LIN {X 0,Y 445.773,Z 444.898,A -85,B 0,C 180,E1 -8709.705,E2 -8709.705} C_VEL
LIN {X 0,Y 445.571,Z 450.254,A -85,B 0,C 180,E1 -8712.561,E2 -8712.561} C_VEL
LIN {X 0,Y 445.558,Z 452.75,A -85,B 0,C 180,E1 -8713.869,E2 -8713.869} C_VEL
LIN {X 0,Y 447.499,Z 463.216,A -85,B 0,C 180,E1 -8714.229,E2 -8714.229} C_VEL
LIN {X 0,Y 449.179,Z 473.492,A -85,B 0,C 180,E1 -8714.691,E2 -8714.691} C_VEL
LIN {X 0,Y 449.183,Z 481.574,A -85,B 0,C 180,E1 -8715.097,E2 -8715.097} C_VEL
LIN {X 0,Y 448.641,Z 491.717,A -85,B 0,C 180,E1 -8715.716,E2 -8715.716} C_VEL
LIN {X 0,Y 448.158,Z 500.718,A -85,B 0,C 180,E1 -8716.395,E2 -8716.395} C_VEL
LIN {X 0,Y 447.767,Z 508.998,A -85,B 0,C 180,E1 -8717.145,E2 -8717.145} C_VEL
LIN {X 0,Y 447.322,Z 516.853,A -85,B 0,C 180,E1 -8717.985,E2 -8717.985} C_VEL
LIN {X 0,Y 446.832,Z 524.074,A -85,B 0,C 180,E1 -8718.891,E2 -8718.891} C_VEL
LIN {X 0,Y 446.495,Z 530.28,A -85,B 0,C 180,E1 -8719.8,E2 -8719.8} C_VEL
LIN {X 0,Y 446.13,Z 536.82,A -85,B 0,C 180,E1 -8720.936,E2 -8720.936} C_VEL
LIN {X 0,Y 445.886,Z 541.323,A -85,B 0,C 180,E1 -8721.845,E2 -8721.845} C_VEL
LIN {X 0,Y 445.655,Z 546.972,A -85,B 0,C 180,E1 -8723.253,E2 -8723.253} C_VEL
LIN {X 0,Y 445.538,Z 551.142,A -85,B 0,C 180,E1 -8724.569,E2 -8724.569} C_VEL
LIN {X 0,Y 445.428,Z 553.506,A -85,B 0,C 180,E1 -8725.475,E2 -8725.475} C_VEL
LIN {X 0,Y 445.387,Z 555.304,A -85,B 0,C 180,E1 -8726.381,E2 -8726.381} C_VEL
LIN {X 0,Y 445.353,Z 557.747,A -85,B 0,C 180,E1 -8728.191,E2 -8728.191} C_VEL
LIN {X 0,Y 445.315,Z 558.334,A -85,B 0,C 180,E1 -8729.096,E2 -8729.096} C_VEL
LIN {X 0,Y 445.315,Z 558.334,A -85,B 0,C 180,E1 -8730.904,E2 -8730.904} C_VEL
LIN {X 0,Y 445.353,Z 557.747,A -85,B 0,C 180,E1 -8731.808,E2 -8731.808} C_VEL
LIN {X 0,Y 445.387,Z 555.305,A -85,B 0,C 180,E1 -8733.619,E2 -8733.619} C_VEL
LIN {X 0,Y 445.5,Z 552.359,A -85,B 0,C 180,E1 -8734.977,E2 -8734.977} C_VEL
LIN {X 0,Y 445.579,Z 548.371,A -85,B 0,C 180,E1 -8736.339,E2 -8736.339} C_VEL
LIN {X 0,Y 445.762,Z 543.24,A -85,B 0,C 180,E1 -8737.701,E2 -8737.701} C_VEL
LIN {X 0,Y 446.078,Z 537.978,A -85,B 0,C 180,E1 -8738.836,E2 -8738.836} C_VEL
LIN {X 0,Y 446.427,Z 531.659,A -85,B 0,C 180,E1 -8739.972,E2 -8739.972} C_VEL
LIN {X 0,Y 446.73,Z 525.704,A -85,B 0,C 180,E1 -8740.882,E2 -8740.882} C_VEL
LIN {X 0,Y 447.175,Z 518.775,A -85,B 0,C 180,E1 -8741.789,E2 -8741.789} C_VEL
LIN {X 0,Y 447.643,Z 510.591,A -85,B 0,C 180,E1 -8742.697,E2 -8742.697} C_VEL
LIN {X 0,Y 448.065,Z 502.329,A -85,B 0,C 180,E1 -8743.47,E2 -8743.47} C_VEL
LIN {X 0,Y 448.563,Z 493.356,A -85,B 0,C 180,E1 -8744.17,E2 -8744.17} C_VEL
LIN {X 0,Y 449.001,Z 484.602,A -85,B 0,C 180,E1 -8744.735,E2 -8744.735} C_VEL
LIN {X 0,Y 449.373,Z 474.797,A -85,B 0,C 180,E1 -8745.244,E2 -8745.244} C_VEL
LIN {X 0,Y 447.738,Z 464.356,A -85,B 0,C 180,E1 -8745.725,E2 -8745.725} C_VEL
LIN {X 0,Y 445.691,Z 453.752,A -85,B 0,C 180,E1 -8746.102,E2 -8746.102} C_VEL
LIN {X 0,Y 445.565,Z 452.689,A -85,B 0,C 180,E1 -8746.163,E2 -8746.163} C_VEL
LIN {X 0,Y 445.699,Z 446.656,A -85,B 0,C 180,E1 -8749.337,E2 -8749.337} C_VEL
LIN {X 0,Y 445.865,Z 441.314,A -85,B 0,C 180,E1 -8752.228,E2 -8752.228} C_VEL
LIN {X 0,Y 446.033,Z 436.032,A -85,B 0,C 180,E1 -8755.177,E2 -8755.177} C_VEL
LIN {X 0,Y 446.267,Z 430.816,A -85,B 0,C 180,E1 -8758.193,E2 -8758.193} C_VEL
LIN {X 0,Y 446.557,Z 424.849,A -85,B 0,C 180,E1 -8761.803,E2 -8761.803} C_VEL
LIN {X 0,Y 446.894,Z 419.658,A -85,B 0,C 180,E1 -8765.137,E2 -8765.137} C_VEL
LIN {X 0,Y 447.24,Z 415.135,A -85,B 0,C 180,E1 -8768.213,E2 -8768.213} C_VEL
LIN {X 0,Y 447.487,Z 410.971,A -85,B 0,C 180,E1 -8771.271,E2 -8771.271} C_VEL
LIN {X 0,Y 447.258,Z 407.884,A -85,B 0,C 180,E1 -8773.74,E2 -8773.74} C_VEL
LIN {X 0,Y 446.793,Z 404.867,A -85,B 0,C 180,E1 -8776.349,E2 -8776.349} C_VEL
LIN {X 0,Y 446.432,Z 402.428,A -85,B 0,C 180,E1 -8778.609,E2 -8778.609} C_VEL
LIN {X 0,Y 446.454,Z 402.376,A -85,B 0,C 180,E1 -8780.974,E2 -8780.974} C_VEL
LIN {X 0,Y 446.418,Z 402.379,A -85,B 0,C 180,E1 -8784.373,E2 -8784.373} C_VEL
LIN {X 0,Y 446.426,Z 402.372,A -85,B 0,C 180,E1 -8787.638,E2 -8787.638} C_VEL
LIN {X 0,Y 446.466,Z 402.374,A -85,B 0,C 180,E1 -8790.791,E2 -8790.791} C_VEL
LIN {X 0,Y 446.473,Z 402.366,A -85,B 0,C 180,E1 -8793.848,E2 -8793.848} C_VEL
LIN {X 0,Y 446.425,Z 402.379,A -85,B 0,C 180,E1 -8796.823,E2 -8796.823} C_VEL
LIN {X 0,Y 446.439,Z 402.37,A -85,B 0,C 180,E1 -8799.736,E2 -8799.736} C_VEL
LIN {X 0,Y 446.459,Z 402.375,A -85,B 0,C 180,E1 -8802.596,E2 -8802.596} C_VEL
LIN {X 0,Y 446.466,Z 402.367,A -85,B 0,C 180,E1 -8805.412,E2 -8805.412} C_VEL
LIN {X 0,Y 446.512,Z 402.364,A -85,B 0,C 180,E1 -8808.192,E2 -8808.192} C_VEL
LIN {X 0,Y 446.594,Z 402.352,A -85,B 0,C 180,E1 -8811.857,E2 -8811.857} C_VEL
LIN {X 0,Y 446.64,Z 402.352,A -85,B 0,C 180,E1 -8814.582,E2 -8814.582} C_VEL
LIN {X 0,Y 446.704,Z 402.337,A -85,B 0,C 180,E1 -8817.294,E2 -8817.294} C_VEL
LIN {X 0,Y 446.787,Z 402.33,A -85,B 0,C 180,E1 -8819.999,E2 -8819.999} C_VEL
LIN {X 0,Y 446.703,Z 402.341,A -85,B 0,C 180,E1 -8822.705,E2 -8822.705} C_VEL
LIN {X 0,Y 446.64,Z 402.353,A -85,B 0,C 180,E1 -8826.323,E2 -8826.323} C_VEL
LIN {X 0,Y 446.531,Z 402.359,A -85,B 0,C 180,E1 -8829.055,E2 -8829.055} C_VEL
LIN {X 0,Y 446.514,Z 402.363,A -85,B 0,C 180,E1 -8832.729,E2 -8832.729} C_VEL
LIN {X 0,Y 446.511,Z 402.368,A -85,B 0,C 180,E1 -8836.238,E2 -8836.238} C_VEL
LIN {X 0,Y 446.461,Z 402.368,A -85,B 0,C 180,E1 -8839.303,E2 -8839.303} C_VEL
LIN {X 0,Y 446.411,Z 402.379,A -85,B 0,C 180,E1 -8842.199,E2 -8842.199} C_VEL
LIN {X 0,Y 446.451,Z 402.369,A -85,B 0,C 180,E1 -8845.152,E2 -8845.152} C_VEL
LIN {X 0,Y 446.477,Z 402.37,A -85,B 0,C 180,E1 -8848.179,E2 -8848.179} C_VEL
LIN {X 0,Y 446.423,Z 402.373,A -85,B 0,C 180,E1 -8851.299,E2 -8851.299} C_VEL
LIN {X 0,Y 446.423,Z 402.373,A -85,B 0,C 180,E1 -8854.523,E2 -8854.523} C_VEL
LIN {X 0,Y 446.431,Z 402.375,A -85,B 0,C 180,E1 -8858.083,E2 -8858.083} C_VEL
LIN {X 0,Y 446.44,Z 402.37,A -85,B 0,C 180,E1 -8860.921,E2 -8860.921} C_VEL
LIN {X 0,Y 446.438,Z 402.376,A -85,B 0,C 180,E1 -8863.841,E2 -8863.841} C_VEL
LIN {X 0,Y 446.44,Z 402.371,A -85,B 0,C 180,E1 -8866.397,E2 -8866.397} C_VEL
LIN {X 0,Y 446.461,Z 402.373,A -85,B 0,C 180,E1 -8869.805,E2 -8869.805} C_VEL
LIN {X 0,Y 446.425,Z 402.374,A -85,B 0,C 180,E1 -8872.124,E2 -8872.124} C_VEL
LIN {X 0,Y 446.425,Z 402.379,A -85,B 0,C 180,E1 -8875.477,E2 -8875.477} C_VEL
LIN {X 0,Y 446.411,Z 402.374,A -85,B 0,C 180,E1 -8878.7,E2 -8878.7} C_VEL
LIN {X 0,Y 446.479,Z 402.368,A -85,B 0,C 180,E1 -8881.822,E2 -8881.822} C_VEL
LIN {X 0,Y 446.453,Z 402.37,A -85,B 0,C 180,E1 -8884.848,E2 -8884.848} C_VEL
LIN {X 0,Y 446.443,Z 402.37,A -85,B 0,C 180,E1 -8888.245,E2 -8888.245} C_VEL
LIN {X 0,Y 446.453,Z 402.374,A -85,B 0,C 180,E1 -8891.65,E2 -8891.65} C_VEL
LIN {X 0,Y 446.503,Z 402.366,A -85,B 0,C 180,E1 -8894.48,E2 -8894.48} C_VEL
LIN {X 0,Y 446.514,Z 402.363,A -85,B 0,C 180,E1 -8898.193,E2 -8898.193} C_VEL
LIN {X 0,Y 446.596,Z 402.355,A -85,B 0,C 180,E1 -8901.858,E2 -8901.858} C_VEL
LIN {X 0,Y 446.644,Z 402.349,A -85,B 0,C 180,E1 -8904.583,E2 -8904.583} C_VEL
LIN {X 0,Y 446.621,Z 402.353,A -85,B 0,C 180,E1 -8907.008,E2 -8907.008} C_VEL
LIN {X 0,Y 446.104,Z 402.421,A -85,B 0,C 180,E1 -8907.761,E2 -8907.761} C_VEL
LIN {X 0,Y 443.287,Z 402.776,A -85,B 0,C 180,E1 -8908.984,E2 -8908.984} C_VEL
LIN {X 0,Y 440.801,Z 403.085,A -85,B 0,C 180,E1 -8909.971,E2 -8909.971} C_VEL
LIN {X 0,Y 439.713,Z 403.216,A -85,B 0,C 180,E1 -8910.734,E2 -8910.734} C_VEL
LIN {X 0,Y 439.618,Z 403.225,A -85,B 0,C 180,E1 -8910.993,E2 -8910.993} C_VEL
LIN {X 0,Y 439.653,Z 403.222,A -85,B 0,C 180,E1 -8912.749,E2 -8912.749} C_VEL
LIN {X 0,Y 439.616,Z 403.227,A -85,B 0,C 180,E1 -8916.425,E2 -8916.425} C_VEL
LIN {X 0,Y 439.497,Z 403.241,A -85,B 0,C 180,E1 -8919.202,E2 -8919.202} C_VEL
LIN {X 0,Y 439.462,Z 403.247,A -85,B 0,C 180,E1 -8922.938,E2 -8922.938} C_VEL
LIN {X 0,Y 439.444,Z 403.247,A -85,B 0,C 180,E1 -8926.349,E2 -8926.349} C_VEL
LIN {X 0,Y 439.399,Z 403.248,A -85,B 0,C 180,E1 -8929.626,E2 -8929.626} C_VEL
LIN {X 0,Y 439.361,Z 403.259,A -85,B 0,C 180,E1 -8932.575,E2 -8932.575} C_VEL
LIN {X 0,Y 439.401,Z 403.247,A -85,B 0,C 180,E1 -8935.585,E2 -8935.585} C_VEL
LIN {X 0,Y 439.413,Z 403.252,A -85,B 0,C 180,E1 -8938.674,E2 -8938.674} C_VEL
LIN {X 0,Y 439.366,Z 403.253,A -85,B 0,C 180,E1 -8942.031,E2 -8942.031} C_VEL
LIN {X 0,Y 439.392,Z 403.248,A -85,B 0,C 180,E1 -8945.341,E2 -8945.341} C_VEL
LIN {X 0,Y 439.391,Z 403.253,A -85,B 0,C 180,E1 -8948.594,E2 -8948.594} C_VEL
LIN {X 0,Y 439.4,Z 403.247,A -85,B 0,C 180,E1 -8951.259,E2 -8951.259} C_VEL
LIN {X 0,Y 439.404,Z 403.249,A -85,B 0,C 180,E1 -8954.728,E2 -8954.728} C_VEL
LIN {X 0,Y 439.391,Z 403.25,A -85,B 0,C 180,E1 -8957.796,E2 -8957.796} C_VEL
LIN {X 0,Y 439.431,Z 403.251,A -85,B 0,C 180,E1 -8960.229,E2 -8960.229} C_VEL
LIN {X 0,Y 439.372,Z 403.253,A -85,B 0,C 180,E1 -8963.713,E2 -8963.713} C_VEL
LIN {X 0,Y 439.37,Z 403.251,A -85,B 0,C 180,E1 -8967.055,E2 -8967.055} C_VEL
LIN {X 0,Y 439.392,Z 403.253,A -85,B 0,C 180,E1 -8970.276,E2 -8970.276} C_VEL
LIN {X 0,Y 439.428,Z 403.246,A -85,B 0,C 180,E1 -8973.589,E2 -8973.589} C_VEL
LIN {X 0,Y 439.382,Z 403.252,A -85,B 0,C 180,E1 -8976.43,E2 -8976.43} C_VEL
LIN {X 0,Y 439.383,Z 403.251,A -85,B 0,C 180,E1 -8979.397,E2 -8979.397} C_VEL
LIN {X 0,Y 439.428,Z 403.246,A -85,B 0,C 180,E1 -8982.31,E2 -8982.31} C_VEL
LIN {X 0,Y 439.447,Z 403.242,A -85,B 0,C 180,E1 -8985.175,E2 -8985.175} C_VEL
LIN {X 0,Y 439.479,Z 403.242,A -85,B 0,C 180,E1 -8988.002,E2 -8988.002} C_VEL
LIN {X 0,Y 439.544,Z 403.237,A -85,B 0,C 180,E1 -8991.727,E2 -8991.727} C_VEL
LIN {X 0,Y 439.617,Z 403.22,A -85,B 0,C 180,E1 -8994.496,E2 -8994.496} C_VEL
LIN {X 0,Y 439.632,Z 403.22,A -85,B 0,C 180,E1 -8998.168,E2 -8998.168} C_VEL
LIN {X 0,Y 439.76,Z 403.205,A -85,B 0,C 180,E1 -9000.001,E2 -9000.001} C_VEL
LIN {X 0,Y 439.653,Z 403.216,A -85,B 0,C 180,E1 -9002.749,E2 -9002.749} C_VEL
LIN {X 0,Y 439.615,Z 403.22,A -85,B 0,C 180,E1 -9006.426,E2 -9006.426} C_VEL
LIN {X 0,Y 439.497,Z 403.239,A -85,B 0,C 180,E1 -9009.202,E2 -9009.202} C_VEL
LIN {X 0,Y 439.463,Z 403.241,A -85,B 0,C 180,E1 -9012.938,E2 -9012.938} C_VEL
LIN {X 0,Y 439.445,Z 403.241,A -85,B 0,C 180,E1 -9016.349,E2 -9016.349} C_VEL
LIN {X 0,Y 439.4,Z 403.251,A -85,B 0,C 180,E1 -9019.627,E2 -9019.627} C_VEL
LIN {X 0,Y 439.363,Z 403.252,A -85,B 0,C 180,E1 -9022.576,E2 -9022.576} C_VEL
LIN {X 0,Y 439.404,Z 403.25,A -85,B 0,C 180,E1 -9025.585,E2 -9025.585} C_VEL
LIN {X 0,Y 439.416,Z 403.247,A -85,B 0,C 180,E1 -9028.674,E2 -9028.674} C_VEL
LIN {X 0,Y 439.369,Z 403.251,A -85,B 0,C 180,E1 -9032.031,E2 -9032.031} C_VEL
LIN {X 0,Y 439.396,Z 403.255,A -85,B 0,C 180,E1 -9035.341,E2 -9035.341} C_VEL
LIN {X 0,Y 439.388,Z 403.256,A -85,B 0,C 180,E1 -9038.595,E2 -9038.595} C_VEL
LIN {X 0,Y 439.381,Z 403.257,A -85,B 0,C 180,E1 -9040.981,E2 -9040.981} C_VEL
LIN {X 0,Y 439.869,Z 406.467,A -85,B 0,C 180,E1 -9044.03,E2 -9044.03} C_VEL
LIN {X 0,Y 440.286,Z 409.495,A -85,B 0,C 180,E1 -9046.656,E2 -9046.656} C_VEL
LIN {X 0,Y 440.456,Z 412.609,A -85,B 0,C 180,E1 -9049.141,E2 -9049.141} C_VEL
LIN {X 0,Y 440.258,Z 415.779,A -85,B 0,C 180,E1 -9051.496,E2 -9051.496} C_VEL
LIN {X 0,Y 439.849,Z 420.662,A -85,B 0,C 180,E1 -9054.886,E2 -9054.886} C_VEL
LIN {X 0,Y 439.508,Z 425.659,A -85,B 0,C 180,E1 -9058.151,E2 -9058.151} C_VEL
LIN {X 0,Y 439.238,Z 430.761,A -85,B 0,C 180,E1 -9061.314,E2 -9061.314} C_VEL
LIN {X 0,Y 438.999,Z 435.948,A -85,B 0,C 180,E1 -9064.39,E2 -9064.39} C_VEL
LIN {X 0,Y 438.794,Z 441.194,A -85,B 0,C 180,E1 -9067.394,E2 -9067.394} C_VEL
LIN {X 0,Y 438.627,Z 446.502,A -85,B 0,C 180,E1 -9070.338,E2 -9070.338} C_VEL
LIN {X 0,Y 438.486,Z 452.562,A -85,B 0,C 180,E1 -9073.599,E2 -9073.599} C_VEL
LIN {X 0,Y 440.489,Z 462.989,A -85,B 0,C 180,E1 -9073.971,E2 -9073.971} C_VEL
LIN {X 0,Y 442.142,Z 473.275,A -85,B 0,C 180,E1 -9074.441,E2 -9074.441} C_VEL
LIN {X 0,Y 442.414,Z 478.317,A -85,B 0,C 180,E1 -9074.687,E2 -9074.687} C_VEL
LIN {X 0,Y 441.855,Z 489.873,A -85,B 0,C 180,E1 -9075.374,E2 -9075.374} C_VEL
LIN {X 0,Y 441.347,Z 499.155,A -85,B 0,C 180,E1 -9076.063,E2 -9076.063} C_VEL
LIN {X 0,Y 440.915,Z 507.557,A -85,B 0,C 180,E1 -9076.815,E2 -9076.815} C_VEL
LIN {X 0,Y 440.353,Z 516.641,A -85,B 0,C 180,E1 -9077.792,E2 -9077.792} C_VEL
LIN {X 0,Y 439.828,Z 523.862,A -85,B 0,C 180,E1 -9078.712,E2 -9078.712} C_VEL
LIN {X 0,Y 439.478,Z 530.068,A -85,B 0,C 180,E1 -9079.636,E2 -9079.636} C_VEL
LIN {X 0,Y 439.085,Z 536.608,A -85,B 0,C 180,E1 -9080.79,E2 -9080.79} C_VEL
LIN {X 0,Y 438.832,Z 541.111,A -85,B 0,C 180,E1 -9081.713,E2 -9081.713} C_VEL
LIN {X 0,Y 438.591,Z 546.604,A -85,B 0,C 180,E1 -9083.097,E2 -9083.097} C_VEL
LIN {X 0,Y 438.439,Z 550.929,A -85,B 0,C 180,E1 -9084.481,E2 -9084.481} C_VEL
LIN {X 0,Y 438.357,Z 553.295,A -85,B 0,C 180,E1 -9085.402,E2 -9085.402} C_VEL
LIN {X 0,Y 438.332,Z 556.48,A -85,B 0,C 180,E1 -9087.243,E2 -9087.243} C_VEL
LIN {X 0,Y 438.275,Z 557.536,A -85,B 0,C 180,E1 -9088.162,E2 -9088.162} C_VEL
LIN {X 0,Y 438.231,Z 558.123,A -85,B 0,C 180,E1 -9089.081,E2 -9089.081} C_VEL
LIN {X 0,Y 438.23,Z 558.123,A -85,B 0,C 180,E1 -9090.919,E2 -9090.919} C_VEL
LIN {X 0,Y 438.275,Z 557.537,A -85,B 0,C 180,E1 -9091.838,E2 -9091.838} C_VEL
LIN {X 0,Y 438.289,Z 555.093,A -85,B 0,C 180,E1 -9093.677,E2 -9093.677} C_VEL
LIN {X 0,Y 438.414,Z 552.147,A -85,B 0,C 180,E1 -9095.058,E2 -9095.058} C_VEL
LIN {X 0,Y 438.507,Z 548.159,A -85,B 0,C 180,E1 -9096.441,E2 -9096.441} C_VEL
LIN {X 0,Y 438.717,Z 543.029,A -85,B 0,C 180,E1 -9097.826,E2 -9097.826} C_VEL
LIN {X 0,Y 439.038,Z 537.766,A -85,B 0,C 180,E1 -9098.979,E2 -9098.979} C_VEL
LIN {X 0,Y 439.4,Z 531.447,A -85,B 0,C 180,E1 -9100.133,E2 -9100.133} C_VEL
LIN {X 0,Y 439.717,Z 525.492,A -85,B 0,C 180,E1 -9101.057,E2 -9101.057} C_VEL
LIN {X 0,Y 440.212,Z 518.563,A -85,B 0,C 180,E1 -9101.978,E2 -9101.978} C_VEL
LIN {X 0,Y 440.697,Z 510.379,A -85,B 0,C 180,E1 -9102.9,E2 -9102.9} C_VEL
LIN {X 0,Y 441.159,Z 501.795,A -85,B 0,C 180,E1 -9103.713,E2 -9103.713} C_VEL
LIN {X 0,Y 441.655,Z 493.144,A -85,B 0,C 180,E1 -9104.397,E2 -9104.397} C_VEL
LIN {X 0,Y 442.161,Z 483.382,A -85,B 0,C 180,E1 -9105.027,E2 -9105.027} C_VEL
LIN {X 0,Y 442.497,Z 475.874,A -85,B 0,C 180,E1 -9105.428,E2 -9105.428} C_VEL
LIN {X 0,Y 440.758,Z 464.605,A -85,B 0,C 180,E1 -9105.964,E2 -9105.964} C_VEL
LIN {X 0,Y 438.726,Z 454.283,A -85,B 0,C 180,E1 -9106.348,E2 -9106.348} C_VEL
LIN {X 0,Y 438.49,Z 452.559,A -85,B 0,C 180,E1 -9106.402,E2 -9106.402} C_VEL
LIN {X 0,Y 438.625,Z 446.5,A -85,B 0,C 180,E1 -9109.662,E2 -9109.662} C_VEL
LIN {X 0,Y 438.793,Z 441.188,A -85,B 0,C 180,E1 -9112.606,E2 -9112.606} C_VEL
LIN {X 0,Y 438.998,Z 435.939,A -85,B 0,C 180,E1 -9115.61,E2 -9115.61} C_VEL
LIN {X 0,Y 439.236,Z 430.751,A -85,B 0,C 180,E1 -9118.686,E2 -9118.686} C_VEL
LIN {X 0,Y 439.527,Z 425.322,A -85,B 0,C 180,E1 -9122.062,E2 -9122.062} C_VEL
LIN {X 0,Y 439.849,Z 420.656,A -85,B 0,C 180,E1 -9125.114,E2 -9125.114} C_VEL
LIN {X 0,Y 440.244,Z 415.74,A -85,B 0,C 180,E1 -9128.534,E2 -9128.534} C_VEL
LIN {X 0,Y 440.459,Z 411.885,A -85,B 0,C 180,E1 -9131.415,E2 -9131.415} C_VEL
LIN {X 0,Y 440.2,Z 408.622,A -85,B 0,C 180,E1 -9134.073,E2 -9134.073} C_VEL
LIN {X 0,Y 439.669,Z 405.005,A -85,B 0,C 180,E1 -9137.331,E2 -9137.331} C_VEL
LIN {X 0,Y 439.379,Z 403.257,A -85,B 0,C 180,E1 -9139.019,E2 -9139.019} C_VEL
LIN {X 0,Y 439.382,Z 403.256,A -85,B 0,C 180,E1 -9141.605,E2 -9141.605} C_VEL
LIN {X 0,Y 439.398,Z 403.255,A -85,B 0,C 180,E1 -9144.843,E2 -9144.843} C_VEL
LIN {X 0,Y 439.386,Z 403.249,A -85,B 0,C 180,E1 -9148.14,E2 -9148.14} C_VEL
LIN {X 0,Y 439.421,Z 403.246,A -85,B 0,C 180,E1 -9151.326,E2 -9151.326} C_VEL
LIN {X 0,Y 439.401,Z 403.25,A -85,B 0,C 180,E1 -9154.414,E2 -9154.414} C_VEL
LIN {X 0,Y 439.36,Z 403.253,A -85,B 0,C 180,E1 -9157.424,E2 -9157.424} C_VEL
LIN {X 0,Y 439.436,Z 403.25,A -85,B 0,C 180,E1 -9160.662,E2 -9160.662} C_VEL
LIN {X 0,Y 439.457,Z 403.243,A -85,B 0,C 180,E1 -9164.224,E2 -9164.224} C_VEL
LIN {X 0,Y 439.478,Z 403.239,A -85,B 0,C 180,E1 -9168.001,E2 -9168.001} C_VEL
LIN {X 0,Y 439.542,Z 403.23,A -85,B 0,C 180,E1 -9171.726,E2 -9171.726} C_VEL
LIN {X 0,Y 439.615,Z 403.228,A -85,B 0,C 180,E1 -9174.495,E2 -9174.495} C_VEL
LIN {X 0,Y 439.63,Z 403.223,A -85,B 0,C 180,E1 -9178.167,E2 -9178.167} C_VEL
LIN {X 0,Y 439.757,Z 403.206,A -85,B 0,C 180,E1 -9179.999,E2 -9179.999} C_VEL
LIN {X 0,Y 439.65,Z 403.219,A -85,B 0,C 180,E1 -9182.748,E2 -9182.748} C_VEL
LIN {X 0,Y 439.611,Z 403.227,A -85,B 0,C 180,E1 -9186.425,E2 -9186.425} C_VEL
LIN {X 0,Y 439.493,Z 403.235,A -85,B 0,C 180,E1 -9189.201,E2 -9189.201} C_VEL
LIN {X 0,Y 439.458,Z 403.24,A -85,B 0,C 180,E1 -9192.937,E2 -9192.937} C_VEL
LIN {X 0,Y 439.453,Z 403.245,A -85,B 0,C 180,E1 -9196.354,E2 -9196.354} C_VEL
LIN {X 0,Y 439.395,Z 403.25,A -85,B 0,C 180,E1 -9199.626,E2 -9199.626} C_VEL
LIN {X 0,Y 439.358,Z 403.254,A -85,B 0,C 180,E1 -9202.575,E2 -9202.575} C_VEL
LIN {X 0,Y 439.398,Z 403.25,A -85,B 0,C 180,E1 -9205.585,E2 -9205.585} C_VEL
LIN {X 0,Y 439.418,Z 403.245,A -85,B 0,C 180,E1 -9208.673,E2 -9208.673} C_VEL
LIN {X 0,Y 439.376,Z 403.256,A -85,B 0,C 180,E1 -9212.033,E2 -9212.033} C_VEL
LIN {X 0,Y 439.389,Z 403.25,A -85,B 0,C 180,E1 -9215.341,E2 -9215.341} C_VEL
LIN {X 0,Y 439.392,Z 403.248,A -85,B 0,C 180,E1 -9218.593,E2 -9218.593} C_VEL
LIN {X 0,Y 439.398,Z 403.249,A -85,B 0,C 180,E1 -9221.259,E2 -9221.259} C_VEL
LIN {X 0,Y 439.403,Z 403.247,A -85,B 0,C 180,E1 -9224.728,E2 -9224.728} C_VEL
LIN {X 0,Y 439.406,Z 403.252,A -85,B 0,C 180,E1 -9227.798,E2 -9227.798} C_VEL
LIN {X 0,Y 439.443,Z 403.243,A -85,B 0,C 180,E1 -9230.23,E2 -9230.23} C_VEL
LIN {X 0,Y 439.371,Z 403.256,A -85,B 0,C 180,E1 -9233.713,E2 -9233.713} C_VEL
LIN {X 0,Y 439.366,Z 403.254,A -85,B 0,C 180,E1 -9237.054,E2 -9237.054} C_VEL
LIN {X 0,Y 439.377,Z 403.25,A -85,B 0,C 180,E1 -9240.274,E2 -9240.274} C_VEL
LIN {X 0,Y 439.425,Z 403.252,A -85,B 0,C 180,E1 -9243.397,E2 -9243.397} C_VEL
LIN {X 0,Y 439.381,Z 403.249,A -85,B 0,C 180,E1 -9246.43,E2 -9246.43} C_VEL
LIN {X 0,Y 439.385,Z 403.256,A -85,B 0,C 180,E1 -9249.397,E2 -9249.397} C_VEL
LIN {X 0,Y 439.427,Z 403.247,A -85,B 0,C 180,E1 -9252.31,E2 -9252.31} C_VEL
LIN {X 0,Y 439.443,Z 403.249,A -85,B 0,C 180,E1 -9255.174,E2 -9255.174} C_VEL
LIN {X 0,Y 439.48,Z 403.239,A -85,B 0,C 180,E1 -9258.002,E2 -9258.002} C_VEL
LIN {X 0,Y 439.544,Z 403.234,A -85,B 0,C 180,E1 -9261.727,E2 -9261.727} C_VEL
LIN {X 0,Y 439.619,Z 403.224,A -85,B 0,C 180,E1 -9264.496,E2 -9264.496} C_VEL
LIN {X 0,Y 439.633,Z 403.222,A -85,B 0,C 180,E1 -9268.168,E2 -9268.168} C_VEL
LIN {X 0,Y 439.761,Z 403.207,A -85,B 0,C 180,E1 -9270,E2 -9270} C_VEL
LIN {X 0,Y 439.618,Z 403.225,A -85,B 0,C 180,E1 -9270.993,E2 -9270.993} C_VEL
LIN {X 0,Y 438.903,Z 403.313,A -85,B 0,C 180,E1 -9271.758,E2 -9271.758} C_VEL
LIN {X 0,Y 435.924,Z 403.686,A -85,B 0,C 180,E1 -9272.997,E2 -9272.997} C_VEL
LIN {X 0,Y 433.473,Z 403.991,A -85,B 0,C 180,E1 -9273.997,E2 -9273.997} C_VEL
LIN {X 0,Y 432.5,Z 404.113,A -85,B 0,C 180,E1 -9274.771,E2 -9274.771} C_VEL
LIN {X 0,Y 432.463,Z 404.114,A -85,B 0,C 180,E1 -9275.033,E2 -9275.033} C_VEL
LIN {X 0,Y 432.582,Z 404.101,A -85,B 0,C 180,E1 -9277.679,E2 -9277.679} C_VEL
LIN {X 0,Y 432.39,Z 404.125,A -85,B 0,C 180,E1 -9281.247,E2 -9281.247} C_VEL
LIN {X 0,Y 432.37,Z 404.127,A -85,B 0,C 180,E1 -9284.112,E2 -9284.112} C_VEL
LIN {X 0,Y 432.394,Z 404.127,A -85,B 0,C 180,E1 -9287.012,E2 -9287.012} C_VEL
LIN {X 0,Y 432.335,Z 404.128,A -85,B 0,C 180,E1 -9289.961,E2 -9289.961} C_VEL
LIN {X 0,Y 432.315,Z 404.133,A -85,B 0,C 180,E1 -9292.964,E2 -9292.964} C_VEL
LIN {X 0,Y 432.36,Z 404.125,A -85,B 0,C 180,E1 -9296.032,E2 -9296.032} C_VEL
LIN {X 0,Y 432.339,Z 404.128,A -85,B 0,C 180,E1 -9299.187,E2 -9299.187} C_VEL
LIN {X 0,Y 432.319,Z 404.136,A -85,B 0,C 180,E1 -9302.443,E2 -9302.443} C_VEL
LIN {X 0,Y 432.341,Z 404.127,A -85,B 0,C 180,E1 -9305.632,E2 -9305.632} C_VEL
LIN {X 0,Y 432.353,Z 404.129,A -85,B 0,C 180,E1 -9308.717,E2 -9308.717} C_VEL
LIN {X 0,Y 432.369,Z 404.124,A -85,B 0,C 180,E1 -9311.792,E2 -9311.792} C_VEL
LIN {X 0,Y 432.374,Z 404.13,A -85,B 0,C 180,E1 -9314.342,E2 -9314.342} C_VEL
LIN {X 0,Y 432.329,Z 404.135,A -85,B 0,C 180,E1 -9318.203,E2 -9318.203} C_VEL
LIN {X 0,Y 432.348,Z 404.126,A -85,B 0,C 180,E1 -9321.284,E2 -9321.284} C_VEL
LIN {X 0,Y 432.34,Z 404.131,A -85,B 0,C 180,E1 -9324.368,E2 -9324.368} C_VEL
LIN {X 0,Y 432.323,Z 404.13,A -85,B 0,C 180,E1 -9327.558,E2 -9327.558} C_VEL
LIN {X 0,Y 432.39,Z 404.124,A -85,B 0,C 180,E1 -9329.744,E2 -9329.744} C_VEL
LIN {X 0,Y 432.395,Z 404.121,A -85,B 0,C 180,E1 -9333.373,E2 -9333.373} C_VEL
LIN {X 0,Y 432.367,Z 404.13,A -85,B 0,C 180,E1 -9336.024,E2 -9336.024} C_VEL
LIN {X 0,Y 432.345,Z 404.126,A -85,B 0,C 180,E1 -9339.046,E2 -9339.046} C_VEL
LIN {X 0,Y 432.374,Z 404.128,A -85,B 0,C 180,E1 -9342.012,E2 -9342.012} C_VEL
LIN {X 0,Y 432.397,Z 404.119,A -85,B 0,C 180,E1 -9344.927,E2 -9344.927} C_VEL
LIN {X 0,Y 432.455,Z 404.12,A -85,B 0,C 180,E1 -9347.804,E2 -9347.804} C_VEL
LIN {X 0,Y 432.488,Z 404.114,A -85,B 0,C 180,E1 -9351.591,E2 -9351.591} C_VEL
LIN {X 0,Y 432.594,Z 404.096,A -85,B 0,C 180,E1 -9354.407,E2 -9354.407} C_VEL
LIN {X 0,Y 432.602,Z 404.096,A -85,B 0,C 180,E1 -9358.139,E2 -9358.139} C_VEL
LIN {X 0,Y 432.73,Z 404.081,A -85,B 0,C 180,E1 -9360.001,E2 -9360.001} C_VEL
LIN {X 0,Y 432.602,Z 404.094,A -85,B 0,C 180,E1 -9362.794,E2 -9362.794} C_VEL
LIN {X 0,Y 432.569,Z 404.098,A -85,B 0,C 180,E1 -9366.531,E2 -9366.531} C_VEL
LIN {X 0,Y 432.44,Z 404.12,A -85,B 0,C 180,E1 -9369.354,E2 -9369.354} C_VEL
LIN {X 0,Y 432.428,Z 404.117,A -85,B 0,C 180,E1 -9372.804,E2 -9372.804} C_VEL
LIN {X 0,Y 432.41,Z 404.118,A -85,B 0,C 180,E1 -9376.48,E2 -9376.48} C_VEL
LIN {X 0,Y 432.336,Z 404.128,A -85,B 0,C 180,E1 -9379.961,E2 -9379.961} C_VEL
LIN {X 0,Y 432.317,Z 404.133,A -85,B 0,C 180,E1 -9382.965,E2 -9382.965} C_VEL
LIN {X 0,Y 432.363,Z 404.124,A -85,B 0,C 180,E1 -9386.033,E2 -9386.033} C_VEL
LIN {X 0,Y 432.341,Z 404.134,A -85,B 0,C 180,E1 -9389.188,E2 -9389.188} C_VEL
LIN {X 0,Y 432.322,Z 404.13,A -85,B 0,C 180,E1 -9392.444,E2 -9392.444} C_VEL
LIN {X 0,Y 432.345,Z 404.131,A -85,B 0,C 180,E1 -9395.633,E2 -9395.633} C_VEL
LIN {X 0,Y 432.351,Z 404.132,A -85,B 0,C 180,E1 -9398.717,E2 -9398.717} C_VEL
LIN {X 0,Y 432.326,Z 404.135,A -85,B 0,C 180,E1 -9400.561,E2 -9400.561} C_VEL
LIN {X 0,Y 432.728,Z 406.574,A -85,B 0,C 180,E1 -9403.043,E2 -9403.043} C_VEL
LIN {X 0,Y 433.178,Z 409.587,A -85,B 0,C 180,E1 -9405.762,E2 -9405.762} C_VEL
LIN {X 0,Y 433.43,Z 412.673,A -85,B 0,C 180,E1 -9408.333,E2 -9408.333} C_VEL
LIN {X 0,Y 433.279,Z 415.81,A -85,B 0,C 180,E1 -9410.758,E2 -9410.758} C_VEL
LIN {X 0,Y 432.873,Z 420.713,A -85,B 0,C 180,E1 -9414.271,E2 -9414.271} C_VEL
LIN {X 0,Y 432.504,Z 425.776,A -85,B 0,C 180,E1 -9417.67,E2 -9417.67} C_VEL
LIN {X 0,Y 432.213,Z 430.694,A -85,B 0,C 180,E1 -9420.803,E2 -9420.803} C_VEL
LIN {X 0,Y 431.979,Z 435.85,A -85,B 0,C 180,E1 -9423.943,E2 -9423.943} C_VEL
LIN {X 0,Y 431.741,Z 441.072,A -85,B 0,C 180,E1 -9427.003,E2 -9427.003} C_VEL
LIN {X 0,Y 431.554,Z 446.345,A -85,B 0,C 180,E1 -9430.002,E2 -9430.002} C_VEL
LIN {X 0,Y 431.399,Z 452.353,A -85,B 0,C 180,E1 -9433.309,E2 -9433.309} C_VEL
LIN {X 0,Y 434.13,Z 467.212,A -85,B 0,C 180,E1 -9433.883,E2 -9433.883} C_VEL
LIN {X 0,Y 435.564,Z 478.106,A -85,B 0,C 180,E1 -9434.44,E2 -9434.44} C_VEL
LIN {X 0,Y 434.956,Z 489.661,A -85,B 0,C 180,E1 -9435.137,E2 -9435.137} C_VEL
LIN {X 0,Y 434.434,Z 498.943,A -85,B 0,C 180,E1 -9435.837,E2 -9435.837} C_VEL
LIN {X 0,Y 433.916,Z 508.134,A -85,B 0,C 180,E1 -9436.681,E2 -9436.681} C_VEL
LIN {X 0,Y 433.398,Z 516.429,A -85,B 0,C 180,E1 -9437.593,E2 -9437.593} C_VEL
LIN {X 0,Y 432.844,Z 523.65,A -85,B 0,C 180,E1 -9438.527,E2 -9438.527} C_VEL
LIN {X 0,Y 432.468,Z 529.855,A -85,B 0,C 180,E1 -9439.466,E2 -9439.466} C_VEL
LIN {X 0,Y 432.059,Z 536.396,A -85,B 0,C 180,E1 -9440.638,E2 -9440.638} C_VEL
LIN {X 0,Y 431.791,Z 540.899,A -85,B 0,C 180,E1 -9441.576,E2 -9441.576} C_VEL
LIN {X 0,Y 431.522,Z 546.393,A -85,B 0,C 180,E1 -9442.984,E2 -9442.984} C_VEL
LIN {X 0,Y 431.343,Z 550.717,A -85,B 0,C 180,E1 -9444.39,E2 -9444.39} C_VEL
LIN {X 0,Y 431.288,Z 553.084,A -85,B 0,C 180,E1 -9445.326,E2 -9445.326} C_VEL
LIN {X 0,Y 431.229,Z 556.269,A -85,B 0,C 180,E1 -9447.197,E2 -9447.197} C_VEL
LIN {X 0,Y 431.2,Z 557.326,A -85,B 0,C 180,E1 -9448.132,E2 -9448.132} C_VEL
LIN {X 0,Y 431.149,Z 557.912,A -85,B 0,C 180,E1 -9449.066,E2 -9449.066} C_VEL
LIN {X 0,Y 431.149,Z 557.913,A -85,B 0,C 180,E1 -9450.934,E2 -9450.934} C_VEL
LIN {X 0,Y 431.2,Z 557.326,A -85,B 0,C 180,E1 -9451.868,E2 -9451.868} C_VEL
LIN {X 0,Y 431.196,Z 554.881,A -85,B 0,C 180,E1 -9453.738,E2 -9453.738} C_VEL
LIN {X 0,Y 431.329,Z 551.936,A -85,B 0,C 180,E1 -9455.141,E2 -9455.141} C_VEL
LIN {X 0,Y 431.442,Z 547.948,A -85,B 0,C 180,E1 -9456.547,E2 -9456.547} C_VEL
LIN {X 0,Y 431.646,Z 542.816,A -85,B 0,C 180,E1 -9457.955,E2 -9457.955} C_VEL
LIN {X 0,Y 431.973,Z 537.553,A -85,B 0,C 180,E1 -9459.127,E2 -9459.127} C_VEL
LIN {X 0,Y 432.362,Z 531.234,A -85,B 0,C 180,E1 -9460.3,E2 -9460.3} C_VEL
LIN {X 0,Y 432.717,Z 525.279,A -85,B 0,C 180,E1 -9461.238,E2 -9461.238} C_VEL
LIN {X 0,Y 433.251,Z 518.352,A -85,B 0,C 180,E1 -9462.174,E2 -9462.174} C_VEL
LIN {X 0,Y 433.76,Z 510.168,A -85,B 0,C 180,E1 -9463.11,E2 -9463.11} C_VEL
LIN {X 0,Y 434.222,Z 501.992,A -85,B 0,C 180,E1 -9463.901,E2 -9463.901} C_VEL
LIN {X 0,Y 434.742,Z 492.931,A -85,B 0,C 180,E1 -9464.631,E2 -9464.631} C_VEL
LIN {X 0,Y 435.284,Z 483.17,A -85,B 0,C 180,E1 -9465.27,E2 -9465.27} C_VEL
LIN {X 0,Y 435.602,Z 476.949,A -85,B 0,C 180,E1 -9465.618,E2 -9465.618} C_VEL
LIN {X 0,Y 433.76,Z 464.865,A -85,B 0,C 180,E1 -9466.213,E2 -9466.213} C_VEL
LIN {X 0,Y 431.558,Z 453.706,A -85,B 0,C 180,E1 -9466.636,E2 -9466.636} C_VEL
LIN {X 0,Y 431.4,Z 452.356,A -85,B 0,C 180,E1 -9466.689,E2 -9466.689} C_VEL
LIN {X 0,Y 431.552,Z 446.344,A -85,B 0,C 180,E1 -9469.998,E2 -9469.998} C_VEL
LIN {X 0,Y 431.74,Z 441.067,A -85,B 0,C 180,E1 -9472.996,E2 -9472.996} C_VEL
LIN {X 0,Y 431.976,Z 435.842,A -85,B 0,C 180,E1 -9476.057,E2 -9476.057} C_VEL
LIN {X 0,Y 432.201,Z 430.687,A -85,B 0,C 180,E1 -9479.197,E2 -9479.197} C_VEL
LIN {X 0,Y 432.511,Z 425.624,A -85,B 0,C 180,E1 -9482.426,E2 -9482.426} C_VEL
LIN {X 0,Y 432.874,Z 420.656,A -85,B 0,C 180,E1 -9485.766,E2 -9485.766} C_VEL
LIN {X 0,Y 433.241,Z 416.325,A -85,B 0,C 180,E1 -9488.862,E2 -9488.862} C_VEL
LIN {X 0,Y 433.421,Z 412.553,A -85,B 0,C 180,E1 -9491.763,E2 -9491.763} C_VEL
LIN {X 0,Y 433.15,Z 409.35,A -85,B 0,C 180,E1 -9494.445,E2 -9494.445} C_VEL
LIN {X 0,Y 432.703,Z 406.549,A -85,B 0,C 180,E1 -9496.986,E2 -9496.986} C_VEL
LIN {X 0,Y 432.324,Z 404.134,A -85,B 0,C 180,E1 -9499.439,E2 -9499.439} C_VEL
LIN {X 0,Y 432.344,Z 404.131,A -85,B 0,C 180,E1 -9501.85,E2 -9501.85} C_VEL
LIN {X 0,Y 432.338,Z 404.134,A -85,B 0,C 180,E1 -9505.322,E2 -9505.322} C_VEL
LIN {X 0,Y 432.331,Z 404.132,A -85,B 0,C 180,E1 -9508.654,E2 -9508.654} C_VEL
LIN {X 0,Y 432.38,Z 404.122,A -85,B 0,C 180,E1 -9511.876,E2 -9511.876} C_VEL
LIN {X 0,Y 432.347,Z 404.13,A -85,B 0,C 180,E1 -9514.998,E2 -9514.998} C_VEL
LIN {X 0,Y 432.352,Z 404.126,A -85,B 0,C 180,E1 -9518.045,E2 -9518.045} C_VEL
LIN {X 0,Y 432.381,Z 404.125,A -85,B 0,C 180,E1 -9521.029,E2 -9521.029} C_VEL
LIN {X 0,Y 432.425,Z 404.117,A -85,B 0,C 180,E1 -9523.96,E2 -9523.96} C_VEL
LIN {X 0,Y 432.453,Z 404.113,A -85,B 0,C 180,E1 -9527.803,E2 -9527.803} C_VEL
LIN {X 0,Y 432.486,Z 404.108,A -85,B 0,C 180,E1 -9531.59,E2 -9531.59} C_VEL
LIN {X 0,Y 432.592,Z 404.102,A -85,B 0,C 180,E1 -9534.406,E2 -9534.406} C_VEL
LIN {X 0,Y 432.6,Z 404.098,A -85,B 0,C 180,E1 -9538.138,E2 -9538.138} C_VEL
LIN {X 0,Y 432.727,Z 404.081,A -85,B 0,C 180,E1 -9539.999,E2 -9539.999} C_VEL
LIN {X 0,Y 432.599,Z 404.097,A -85,B 0,C 180,E1 -9542.793,E2 -9542.793} C_VEL
LIN {X 0,Y 432.566,Z 404.103,A -85,B 0,C 180,E1 -9546.53,E2 -9546.53} C_VEL
LIN {X 0,Y 432.436,Z 404.115,A -85,B 0,C 180,E1 -9549.353,E2 -9549.353} C_VEL
LIN {X 0,Y 432.423,Z 404.117,A -85,B 0,C 180,E1 -9552.803,E2 -9552.803} C_VEL
LIN {X 0,Y 432.415,Z 404.12,A -85,B 0,C 180,E1 -9556.483,E2 -9556.483} C_VEL
LIN {X 0,Y 432.331,Z 404.134,A -85,B 0,C 180,E1 -9559.96,E2 -9559.96} C_VEL
LIN {X 0,Y 432.312,Z 404.13,A -85,B 0,C 180,E1 -9562.964,E2 -9562.964} C_VEL
LIN {X 0,Y 432.358,Z 404.132,A -85,B 0,C 180,E1 -9566.032,E2 -9566.032} C_VEL
LIN {X 0,Y 432.345,Z 404.126,A -85,B 0,C 180,E1 -9569.187,E2 -9569.187} C_VEL
LIN {X 0,Y 432.324,Z 404.131,A -85,B 0,C 180,E1 -9572.295,E2 -9572.295} C_VEL
LIN {X 0,Y 432.333,Z 404.128,A -85,B 0,C 180,E1 -9574.677,E2 -9574.677} C_VEL
LIN {X 0,Y 432.346,Z 404.129,A -85,B 0,C 180,E1 -9578.148,E2 -9578.148} C_VEL
LIN {X 0,Y 432.366,Z 404.129,A -85,B 0,C 180,E1 -9581.608,E2 -9581.608} C_VEL
LIN {X 0,Y 432.371,Z 404.124,A -85,B 0,C 180,E1 -9584.342,E2 -9584.342} C_VEL
LIN {X 0,Y 432.359,Z 404.125,A -85,B 0,C 180,E1 -9587.009,E2 -9587.009} C_VEL
LIN {X 0,Y 432.35,Z 404.13,A -85,B 0,C 180,E1 -9589.817,E2 -9589.817} C_VEL
LIN {X 0,Y 432.31,Z 404.132,A -85,B 0,C 180,E1 -9593.023,E2 -9593.023} C_VEL
LIN {X 0,Y 432.354,Z 404.127,A -85,B 0,C 180,E1 -9595.997,E2 -9595.997} C_VEL
LIN {X 0,Y 432.342,Z 404.134,A -85,B 0,C 180,E1 -9599.49,E2 -9599.49} C_VEL
LIN {X 0,Y 432.388,Z 404.123,A -85,B 0,C 180,E1 -9602.929,E2 -9602.929} C_VEL
LIN {X 0,Y 432.366,Z 404.124,A -85,B 0,C 180,E1 -9606.024,E2 -9606.024} C_VEL
LIN {X 0,Y 432.346,Z 404.13,A -85,B 0,C 180,E1 -9609.046,E2 -9609.046} C_VEL
LIN {X 0,Y 432.374,Z 404.126,A -85,B 0,C 180,E1 -9612.011,E2 -9612.011} C_VEL
LIN {X 0,Y 432.391,Z 404.127,A -85,B 0,C 180,E1 -9614.927,E2 -9614.927} C_VEL
LIN {X 0,Y 432.455,Z 404.115,A -85,B 0,C 180,E1 -9617.804,E2 -9617.804} C_VEL
LIN {X 0,Y 432.488,Z 404.113,A -85,B 0,C 180,E1 -9621.591,E2 -9621.591} C_VEL
LIN {X 0,Y 432.595,Z 404.099,A -85,B 0,C 180,E1 -9624.406,E2 -9624.406} C_VEL
LIN {X 0,Y 432.603,Z 404.097,A -85,B 0,C 180,E1 -9628.138,E2 -9628.138} C_VEL
LIN {X 0,Y 432.73,Z 404.083,A -85,B 0,C 180,E1 -9630,E2 -9630} C_VEL
LIN {X 0,Y 432.602,Z 404.1,A -85,B 0,C 180,E1 -9632.794,E2 -9632.794} C_VEL
LIN {X 0,Y 432.463,Z 404.114,A -85,B 0,C 180,E1 -9635.033,E2 -9635.033} C_VEL
LIN {X 0,Y 431.904,Z 404.185,A -85,B 0,C 180,E1 -9635.812,E2 -9635.812} C_VEL
LIN {X 0,Y 429.057,Z 404.542,A -85,B 0,C 180,E1 -9637.077,E2 -9637.077} C_VEL
LIN {X 0,Y 426.572,Z 404.85,A -85,B 0,C 180,E1 -9638.098,E2 -9638.098} C_VEL
LIN {X 0,Y 425.49,Z 404.987,A -85,B 0,C 180,E1 -9638.888,E2 -9638.888} C_VEL
LIN {X 0,Y 425.399,Z 404.995,A -85,B 0,C 180,E1 -9639.156,E2 -9639.156} C_VEL
LIN {X 0,Y 425.39,Z 405,A -85,B 0,C 180,E1 -9642.904,E2 -9642.904} C_VEL
LIN {X 0,Y 425.358,Z 405.003,A -85,B 0,C 180,E1 -9646.605,E2 -9646.605} C_VEL
LIN {X 0,Y 425.325,Z 405.002,A -85,B 0,C 180,E1 -9649.636,E2 -9649.636} C_VEL
LIN {X 0,Y 425.303,Z 405.004,A -85,B 0,C 180,E1 -9653.365,E2 -9653.365} C_VEL
LIN {X 0,Y 425.345,Z 405.002,A -85,B 0,C 180,E1 -9656.845,E2 -9656.845} C_VEL
LIN {X 0,Y 425.287,Z 405.005,A -85,B 0,C 180,E1 -9659.72,E2 -9659.72} C_VEL
LIN {X 0,Y 425.278,Z 405.008,A -85,B 0,C 180,E1 -9663.048,E2 -9663.048} C_VEL
LIN {X 0,Y 425.281,Z 405.008,A -85,B 0,C 180,E1 -9665.929,E2 -9665.929} C_VEL
LIN {X 0,Y 425.306,Z 405.004,A -85,B 0,C 180,E1 -9669.046,E2 -9669.046} C_VEL
LIN {X 0,Y 425.327,Z 405.004,A -85,B 0,C 180,E1 -9672.646,E2 -9672.646} C_VEL
LIN {X 0,Y 425.29,Z 405.005,A -85,B 0,C 180,E1 -9675.282,E2 -9675.282} C_VEL
LIN {X 0,Y 425.27,Z 405.01,A -85,B 0,C 180,E1 -9678.622,E2 -9678.622} C_VEL
LIN {X 0,Y 425.31,Z 405.002,A -85,B 0,C 180,E1 -9681.103,E2 -9681.103} C_VEL
LIN {X 0,Y 425.295,Z 405.006,A -85,B 0,C 180,E1 -9684.664,E2 -9684.664} C_VEL
LIN {X 0,Y 425.269,Z 405.015,A -85,B 0,C 180,E1 -9688.074,E2 -9688.074} C_VEL
LIN {X 0,Y 425.333,Z 405,A -85,B 0,C 180,E1 -9691.369,E2 -9691.369} C_VEL
LIN {X 0,Y 425.291,Z 405.006,A -85,B 0,C 180,E1 -9694.555,E2 -9694.555} C_VEL
LIN {X 0,Y 425.283,Z 405.009,A -85,B 0,C 180,E1 -9697.662,E2 -9697.662} C_VEL
LIN {X 0,Y 425.357,Z 404.997,A -85,B 0,C 180,E1 -9700.704,E2 -9700.704} C_VEL
LIN {X 0,Y 425.394,Z 404.997,A -85,B 0,C 180,E1 -9703.689,E2 -9703.689} C_VEL
LIN {X 0,Y 425.407,Z 404.995,A -85,B 0,C 180,E1 -9707.599,E2 -9707.599} C_VEL
LIN {X 0,Y 425.438,Z 404.99,A -85,B 0,C 180,E1 -9711.45,E2 -9711.45} C_VEL
LIN {X 0,Y 425.55,Z 404.974,A -85,B 0,C 180,E1 -9714.314,E2 -9714.314} C_VEL
LIN {X 0,Y 425.572,Z 404.972,A -85,B 0,C 180,E1 -9718.108,E2 -9718.108} C_VEL
LIN {X 0,Y 425.699,Z 404.957,A -85,B 0,C 180,E1 -9720.001,E2 -9720.001} C_VEL
LIN {X 0,Y 425.554,Z 404.972,A -85,B 0,C 180,E1 -9722.84,E2 -9722.84} C_VEL
LIN {X 0,Y 425.528,Z 404.975,A -85,B 0,C 180,E1 -9726.639,E2 -9726.639} C_VEL
LIN {X 0,Y 425.398,Z 404.998,A -85,B 0,C 180,E1 -9729.51,E2 -9729.51} C_VEL
LIN {X 0,Y 425.391,Z 404.994,A -85,B 0,C 180,E1 -9732.904,E2 -9732.904} C_VEL
LIN {X 0,Y 425.359,Z 404.997,A -85,B 0,C 180,E1 -9736.606,E2 -9736.606} C_VEL
LIN {X 0,Y 425.326,Z 405.004,A -85,B 0,C 180,E1 -9739.636,E2 -9739.636} C_VEL
LIN {X 0,Y 425.305,Z 405.009,A -85,B 0,C 180,E1 -9743.366,E2 -9743.366} C_VEL
LIN {X 0,Y 425.346,Z 405.001,A -85,B 0,C 180,E1 -9746.845,E2 -9746.845} C_VEL
LIN {X 0,Y 425.29,Z 405.006,A -85,B 0,C 180,E1 -9749.72,E2 -9749.72} C_VEL
LIN {X 0,Y 425.281,Z 405.013,A -85,B 0,C 180,E1 -9753.049,E2 -9753.049} C_VEL
LIN {X 0,Y 425.284,Z 405.009,A -85,B 0,C 180,E1 -9755.93,E2 -9755.93} C_VEL
LIN {X 0,Y 425.3,Z 405.011,A -85,B 0,C 180,E1 -9759.044,E2 -9759.044} C_VEL
LIN {X 0,Y 425.33,Z 405.23,A -85,B 0,C 180,E1 -9760.529,E2 -9760.529} C_VEL
LIN {X 0,Y 425.83,Z 408.662,A -85,B 0,C 180,E1 -9763.883,E2 -9763.883} C_VEL
LIN {X 0,Y 426.258,Z 411.566,A -85,B 0,C 180,E1 -9766.507,E2 -9766.507} C_VEL
LIN {X 0,Y 426.383,Z 414.966,A -85,B 0,C 180,E1 -9769.307,E2 -9769.307} C_VEL
LIN {X 0,Y 426.075,Z 419.058,A -85,B 0,C 180,E1 -9772.389,E2 -9772.389} C_VEL
LIN {X 0,Y 425.681,Z 423.945,A -85,B 0,C 180,E1 -9775.852,E2 -9775.852} C_VEL
LIN {X 0,Y 425.297,Z 429.024,A -85,B 0,C 180,E1 -9779.238,E2 -9779.238} C_VEL
LIN {X 0,Y 425.025,Z 434.039,A -85,B 0,C 180,E1 -9782.42,E2 -9782.42} C_VEL
LIN {X 0,Y 424.778,Z 439.212,A -85,B 0,C 180,E1 -9785.567,E2 -9785.567} C_VEL
LIN {X 0,Y 424.592,Z 444.453,A -85,B 0,C 180,E1 -9788.645,E2 -9788.645} C_VEL
LIN {X 0,Y 424.367,Z 449.712,A -85,B 0,C 180,E1 -9791.66,E2 -9791.66} C_VEL
LIN {X 0,Y 424.329,Z 452.422,A -85,B 0,C 180,E1 -9793.048,E2 -9793.048} C_VEL
LIN {X 0,Y 426.272,Z 462.585,A -85,B 0,C 180,E1 -9793.423,E2 -9793.423} C_VEL
LIN {X 0,Y 428.062,Z 472.839,A -85,B 0,C 180,E1 -9793.915,E2 -9793.915} C_VEL
LIN {X 0,Y 428.657,Z 478.922,A -85,B 0,C 180,E1 -9794.244,E2 -9794.244} C_VEL
LIN {X 0,Y 428.082,Z 489.449,A -85,B 0,C 180,E1 -9794.893,E2 -9794.893} C_VEL
LIN {X 0,Y 427.54,Z 498.731,A -85,B 0,C 180,E1 -9795.604,E2 -9795.604} C_VEL
LIN {X 0,Y 427.059,Z 506.726,A -85,B 0,C 180,E1 -9796.335,E2 -9796.335} C_VEL
LIN {X 0,Y 426.591,Z 514.297,A -85,B 0,C 180,E1 -9797.149,E2 -9797.149} C_VEL
LIN {X 0,Y 425.872,Z 523.438,A -85,B 0,C 180,E1 -9798.337,E2 -9798.337} C_VEL
LIN {X 0,Y 425.454,Z 529.643,A -85,B 0,C 180,E1 -9799.29,E2 -9799.29} C_VEL
LIN {X 0,Y 425.025,Z 536.184,A -85,B 0,C 180,E1 -9800.482,E2 -9800.482} C_VEL
LIN {X 0,Y 424.737,Z 540.687,A -85,B 0,C 180,E1 -9801.436,E2 -9801.436} C_VEL
LIN {X 0,Y 424.44,Z 546.18,A -85,B 0,C 180,E1 -9802.866,E2 -9802.866} C_VEL
LIN {X 0,Y 424.252,Z 550.505,A -85,B 0,C 180,E1 -9804.296,E2 -9804.296} C_VEL
LIN {X 0,Y 424.219,Z 552.873,A -85,B 0,C 180,E1 -9805.248,E2 -9805.248} C_VEL
LIN {X 0,Y 424.126,Z 556.057,A -85,B 0,C 180,E1 -9807.15,E2 -9807.15} C_VEL
LIN {X 0,Y 424.126,Z 557.115,A -85,B 0,C 180,E1 -9808.101,E2 -9808.101} C_VEL
LIN {X 0,Y 424.07,Z 557.702,A -85,B 0,C 180,E1 -9809.05,E2 -9809.05} C_VEL
LIN {X 0,Y 424.07,Z 557.702,A -85,B 0,C 180,E1 -9810.949,E2 -9810.949} C_VEL
LIN {X 0,Y 424.126,Z 557.115,A -85,B 0,C 180,E1 -9811.899,E2 -9811.899} C_VEL
LIN {X 0,Y 424.108,Z 554.67,A -85,B 0,C 180,E1 -9813.8,E2 -9813.8} C_VEL
LIN {X 0,Y 424.246,Z 551.724,A -85,B 0,C 180,E1 -9815.227,E2 -9815.227} C_VEL
LIN {X 0,Y 424.361,Z 547.735,A -85,B 0,C 180,E1 -9816.657,E2 -9816.657} C_VEL
LIN {X 0,Y 424.59,Z 542.604,A -85,B 0,C 180,E1 -9818.088,E2 -9818.088} C_VEL
LIN {X 0,Y 424.925,Z 537.341,A -85,B 0,C 180,E1 -9819.28,E2 -9819.28} C_VEL
LIN {X 0,Y 425.336,Z 531.021,A -85,B 0,C 180,E1 -9820.472,E2 -9820.472} C_VEL
LIN {X 0,Y 425.732,Z 525.067,A -85,B 0,C 180,E1 -9821.425,E2 -9821.425} C_VEL
LIN {X 0,Y 426.3,Z 518.14,A -85,B 0,C 180,E1 -9822.375,E2 -9822.375} C_VEL
LIN {X 0,Y 426.822,Z 509.955,A -85,B 0,C 180,E1 -9823.327,E2 -9823.327} C_VEL
LIN {X 0,Y 427.339,Z 501.171,A -85,B 0,C 180,E1 -9824.184,E2 -9824.184} C_VEL
LIN {X 0,Y 427.871,Z 492.72,A -85,B 0,C 180,E1 -9824.871,E2 -9824.871} C_VEL
LIN {X 0,Y 428.441,Z 482.959,A -85,B 0,C 180,E1 -9825.52,E2 -9825.52} C_VEL
LIN {X 0,Y 428.572,Z 476.731,A -85,B 0,C 180,E1 -9825.881,E2 -9825.881} C_VEL
LIN {X 0,Y 426.631,Z 464.259,A -85,B 0,C 180,E1 -9826.505,E2 -9826.505} C_VEL
LIN {X 0,Y 424.479,Z 453.446,A -85,B 0,C 180,E1 -9826.922,E2 -9826.922} C_VEL
LIN {X 0,Y 424.317,Z 452.163,A -85,B 0,C 180,E1 -9826.981,E2 -9826.981} C_VEL
LIN {X 0,Y 424.505,Z 446.189,A -85,B 0,C 180,E1 -9830.344,E2 -9830.344} C_VEL
LIN {X 0,Y 424.679,Z 440.94,A -85,B 0,C 180,E1 -9833.401,E2 -9833.401} C_VEL
LIN {X 0,Y 424.968,Z 435.38,A -85,B 0,C 180,E1 -9836.742,E2 -9836.742} C_VEL
LIN {X 0,Y 425.188,Z 430.627,A -85,B 0,C 180,E1 -9839.727,E2 -9839.727} C_VEL
LIN {X 0,Y 425.509,Z 425.589,A -85,B 0,C 180,E1 -9843.027,E2 -9843.027} C_VEL
LIN {X 0,Y 425.851,Z 421.235,A -85,B 0,C 180,E1 -9846.033,E2 -9846.033} C_VEL
LIN {X 0,Y 426.254,Z 416.913,A -85,B 0,C 180,E1 -9849.201,E2 -9849.201} C_VEL
LIN {X 0,Y 426.375,Z 413.193,A -85,B 0,C 180,E1 -9852.119,E2 -9852.119} C_VEL
LIN {X 0,Y 426.06,Z 410.07,A -85,B 0,C 180,E1 -9854.821,E2 -9854.821} C_VEL
LIN {X 0,Y 425.523,Z 406.683,A -85,B 0,C 180,E1 -9858.006,E2 -9858.006} C_VEL
LIN {X 0,Y 425.288,Z 405.012,A -85,B 0,C 180,E1 -9859.872,E2 -9859.872} C_VEL
LIN {X 0,Y 425.282,Z 405.012,A -85,B 0,C 180,E1 -9862.486,E2 -9862.486} C_VEL
LIN {X 0,Y 425.305,Z 405.005,A -85,B 0,C 180,E1 -9865.817,E2 -9865.817} C_VEL
LIN {X 0,Y 425.302,Z 405.006,A -85,B 0,C 180,E1 -9869.235,E2 -9869.235} C_VEL
LIN {X 0,Y 425.346,Z 405.001,A -85,B 0,C 180,E1 -9872.442,E2 -9872.442} C_VEL
LIN {X 0,Y 425.347,Z 404.998,A -85,B 0,C 180,E1 -9875.601,E2 -9875.601} C_VEL
LIN {X 0,Y 425.288,Z 405.012,A -85,B 0,C 180,E1 -9878.681,E2 -9878.681} C_VEL
LIN {X 0,Y 425.328,Z 405,A -85,B 0,C 180,E1 -9881.702,E2 -9881.702} C_VEL
LIN {X 0,Y 425.344,Z 405.005,A -85,B 0,C 180,E1 -9884.67,E2 -9884.67} C_VEL
LIN {X 0,Y 425.406,Z 404.99,A -85,B 0,C 180,E1 -9887.598,E2 -9887.598} C_VEL
LIN {X 0,Y 425.436,Z 404.987,A -85,B 0,C 180,E1 -9891.449,E2 -9891.449} C_VEL
LIN {X 0,Y 425.548,Z 404.978,A -85,B 0,C 180,E1 -9894.313,E2 -9894.313} C_VEL
LIN {X 0,Y 425.569,Z 404.974,A -85,B 0,C 180,E1 -9898.107,E2 -9898.107} C_VEL
LIN {X 0,Y 425.696,Z 404.957,A -85,B 0,C 180,E1 -9899.999,E2 -9899.999} C_VEL
LIN {X 0,Y 425.551,Z 404.974,A -85,B 0,C 180,E1 -9902.839,E2 -9902.839} C_VEL
LIN {X 0,Y 425.524,Z 404.979,A -85,B 0,C 180,E1 -9906.638,E2 -9906.638} C_VEL
LIN {X 0,Y 425.394,Z 404.992,A -85,B 0,C 180,E1 -9909.509,E2 -9909.509} C_VEL
LIN {X 0,Y 425.386,Z 404.993,A -85,B 0,C 180,E1 -9912.903,E2 -9912.903} C_VEL
LIN {X 0,Y 425.363,Z 404.998,A -85,B 0,C 180,E1 -9916.609,E2 -9916.609} C_VEL
LIN {X 0,Y 425.321,Z 405.003,A -85,B 0,C 180,E1 -9919.635,E2 -9919.635} C_VEL
LIN {X 0,Y 425.3,Z 405.004,A -85,B 0,C 180,E1 -9923.365,E2 -9923.365} C_VEL
LIN {X 0,Y 425.341,Z 404.999,A -85,B 0,C 180,E1 -9926.844,E2 -9926.844} C_VEL
LIN {X 0,Y 425.311,Z 405.007,A -85,B 0,C 180,E1 -9929.717,E2 -9929.717} C_VEL
LIN {X 0,Y 425.277,Z 405.007,A -85,B 0,C 180,E1 -9933.048,E2 -9933.048} C_VEL
LIN {X 0,Y 425.277,Z 405.013,A -85,B 0,C 180,E1 -9935.929,E2 -9935.929} C_VEL
LIN {X 0,Y 425.306,Z 405.003,A -85,B 0,C 180,E1 -9939.046,E2 -9939.046} C_VEL
LIN {X 0,Y 425.325,Z 405.001,A -85,B 0,C 180,E1 -9942.646,E2 -9942.646} C_VEL
LIN {X 0,Y 425.312,Z 405.005,A -85,B 0,C 180,E1 -9946.052,E2 -9946.052} C_VEL
LIN {X 0,Y 425.303,Z 405.003,A -85,B 0,C 180,E1 -9948.626,E2 -9948.626} C_VEL
LIN {X 0,Y 425.315,Z 405.004,A -85,B 0,C 180,E1 -9951.104,E2 -9951.104} C_VEL
LIN {X 0,Y 425.294,Z 405.004,A -85,B 0,C 180,E1 -9954.664,E2 -9954.664} C_VEL
LIN {X 0,Y 425.259,Z 405.01,A -85,B 0,C 180,E1 -9958.073,E2 -9958.073} C_VEL
LIN {X 0,Y 425.326,Z 405.007,A -85,B 0,C 180,E1 -9961.368,E2 -9961.368} C_VEL
LIN {X 0,Y 425.29,Z 405.005,A -85,B 0,C 180,E1 -9964.555,E2 -9964.555} C_VEL
LIN {X 0,Y 425.283,Z 405.009,A -85,B 0,C 180,E1 -9967.662,E2 -9967.662} C_VEL
LIN {X 0,Y 425.357,Z 404.998,A -85,B 0,C 180,E1 -9970.704,E2 -9970.704} C_VEL
LIN {X 0,Y 425.384,Z 404.998,A -85,B 0,C 180,E1 -9973.689,E2 -9973.689} C_VEL
LIN {X 0,Y 425.408,Z 404.994,A -85,B 0,C 180,E1 -9977.598,E2 -9977.598} C_VEL
LIN {X 0,Y 425.439,Z 404.992,A -85,B 0,C 180,E1 -9981.45,E2 -9981.45} C_VEL
LIN {X 0,Y 425.552,Z 404.976,A -85,B 0,C 180,E1 -9984.314,E2 -9984.314} C_VEL
LIN {X 0,Y 425.572,Z 404.973,A -85,B 0,C 180,E1 -9988.107,E2 -9988.107} C_VEL
LIN {X 0,Y 425.7,Z 404.959,A -85,B 0,C 180,E1 -9990,E2 -9990} C_VEL
LIN {X 0,Y 425.554,Z 404.978,A -85,B 0,C 180,E1 -9992.84,E2 -9992.84} C_VEL
LIN {X 0,Y 425.529,Z 404.981,A -85,B 0,C 180,E1 -9996.639,E2 -9996.639} C_VEL
LIN {X 0,Y 425.399,Z 404.995,A -85,B 0,C 180,E1 -9999.156,E2 -9999.156} C_VEL
LIN {X 0,Y 424.728,Z 405.081,A -85,B 0,C 180,E1 -9999.946,E2 -9999.946} C_VEL
LIN {X 0,Y 421.879,Z 405.438,A -85,B 0,C 180,E1 -10001.229,E2 -10001.229} C_VEL
LIN {X 0,Y 419.463,Z 405.739,A -85,B 0,C 180,E1 -10002.265,E2 -10002.265} C_VEL
LIN {X 0,Y 418.412,Z 405.869,A -85,B 0,C 180,E1 -10003.066,E2 -10003.066} C_VEL
LIN {X 0,Y 418.318,Z 405.878,A -85,B 0,C 180,E1 -10003.337,E2 -10003.337} C_VEL
LIN {X 0,Y 418.309,Z 405.882,A -85,B 0,C 180,E1 -10006.736,E2 -10006.736} C_VEL
LIN {X 0,Y 418.267,Z 405.881,A -85,B 0,C 180,E1 -10009.791,E2 -10009.791} C_VEL
LIN {X 0,Y 418.234,Z 405.89,A -85,B 0,C 180,E1 -10012.736,E2 -10012.736} C_VEL
LIN {X 0,Y 418.267,Z 405.88,A -85,B 0,C 180,E1 -10015.904,E2 -10015.904} C_VEL
LIN {X 0,Y 418.261,Z 405.882,A -85,B 0,C 180,E1 -10019.162,E2 -10019.162} C_VEL
LIN {X 0,Y 418.253,Z 405.885,A -85,B 0,C 180,E1 -10022.844,E2 -10022.844} C_VEL
LIN {X 0,Y 418.244,Z 405.887,A -85,B 0,C 180,E1 -10026.239,E2 -10026.239} C_VEL
LIN {X 0,Y 418.26,Z 405.881,A -85,B 0,C 180,E1 -10029.68,E2 -10029.68} C_VEL
LIN {X 0,Y 418.281,Z 405.885,A -85,B 0,C 180,E1 -10032.33,E2 -10032.33} C_VEL
LIN {X 0,Y 418.246,Z 405.883,A -85,B 0,C 180,E1 -10035.111,E2 -10035.111} C_VEL
LIN {X 0,Y 418.235,Z 405.886,A -85,B 0,C 180,E1 -10037.767,E2 -10037.767} C_VEL
LIN {X 0,Y 418.255,Z 405.884,A -85,B 0,C 180,E1 -10040.618,E2 -10040.618} C_VEL
LIN {X 0,Y 418.241,Z 405.888,A -85,B 0,C 180,E1 -10043.976,E2 -10043.976} C_VEL
LIN {X 0,Y 418.255,Z 405.881,A -85,B 0,C 180,E1 -10047.156,E2 -10047.156} C_VEL
LIN {X 0,Y 418.27,Z 405.88,A -85,B 0,C 180,E1 -10050.839,E2 -10050.839} C_VEL
LIN {X 0,Y 418.266,Z 405.886,A -85,B 0,C 180,E1 -10054.096,E2 -10054.096} C_VEL
LIN {X 0,Y 418.233,Z 405.885,A -85,B 0,C 180,E1 -10057.264,E2 -10057.264} C_VEL
LIN {X 0,Y 418.278,Z 405.881,A -85,B 0,C 180,E1 -10060.365,E2 -10060.365} C_VEL
LIN {X 0,Y 418.322,Z 405.875,A -85,B 0,C 180,E1 -10063.405,E2 -10063.405} C_VEL
LIN {X 0,Y 418.342,Z 405.871,A -85,B 0,C 180,E1 -10067,E2 -10067} C_VEL
LIN {X 0,Y 418.337,Z 405.872,A -85,B 0,C 180,E1 -10070.329,E2 -10070.329} C_VEL
LIN {X 0,Y 418.509,Z 405.851,A -85,B 0,C 180,E1 -10072.28,E2 -10072.28} C_VEL
LIN {X 0,Y 418.509,Z 405.851,A -85,B 0,C 180,E1 -10074.218,E2 -10074.218} C_VEL
LIN {X 0,Y 418.541,Z 405.848,A -85,B 0,C 180,E1 -10078.076,E2 -10078.076} C_VEL
LIN {X 0,Y 418.669,Z 405.832,A -85,B 0,C 180,E1 -10080.001,E2 -10080.001} C_VEL
LIN {X 0,Y 418.508,Z 405.85,A -85,B 0,C 180,E1 -10082.888,E2 -10082.888} C_VEL
LIN {X 0,Y 418.491,Z 405.852,A -85,B 0,C 180,E1 -10086.752,E2 -10086.752} C_VEL
LIN {X 0,Y 418.397,Z 405.864,A -85,B 0,C 180,E1 -10088.696,E2 -10088.696} C_VEL
LIN {X 0,Y 418.313,Z 405.879,A -85,B 0,C 180,E1 -10091.632,E2 -10091.632} C_VEL
LIN {X 0,Y 418.301,Z 405.876,A -85,B 0,C 180,E1 -10094.598,E2 -10094.598} C_VEL
LIN {X 0,Y 418.286,Z 405.881,A -85,B 0,C 180,E1 -10097.604,E2 -10097.604} C_VEL
LIN {X 0,Y 418.248,Z 405.883,A -85,B 0,C 180,E1 -10100.664,E2 -10100.664} C_VEL
LIN {X 0,Y 418.286,Z 405.879,A -85,B 0,C 180,E1 -10103.782,E2 -10103.782} C_VEL
LIN {X 0,Y 418.309,Z 405.88,A -85,B 0,C 180,E1 -10107.071,E2 -10107.071} C_VEL
LIN {X 0,Y 418.243,Z 405.883,A -85,B 0,C 180,E1 -10110.273,E2 -10110.273} C_VEL
LIN {X 0,Y 418.248,Z 405.886,A -85,B 0,C 180,E1 -10113.678,E2 -10113.678} C_VEL
LIN {X 0,Y 418.245,Z 405.889,A -85,B 0,C 180,E1 -10117.224,E2 -10117.224} C_VEL
LIN {X 0,Y 418.252,Z 405.888,A -85,B 0,C 180,E1 -10119.682,E2 -10119.682} C_VEL
LIN {X 0,Y 418.608,Z 408.263,A -85,B 0,C 180,E1 -10122.379,E2 -10122.379} C_VEL
LIN {X 0,Y 419.067,Z 411.242,A -85,B 0,C 180,E1 -10125.222,E2 -10125.222} C_VEL
LIN {X 0,Y 419.382,Z 414.322,A -85,B 0,C 180,E1 -10127.909,E2 -10127.909} C_VEL
LIN {X 0,Y 419.28,Z 417.486,A -85,B 0,C 180,E1 -10130.449,E2 -10130.449} C_VEL
LIN {X 0,Y 418.87,Z 421.745,A -85,B 0,C 180,E1 -10133.646,E2 -10133.646} C_VEL
LIN {X 0,Y 418.449,Z 426.678,A -85,B 0,C 180,E1 -10137.116,E2 -10137.116} C_VEL
LIN {X 0,Y 418.178,Z 430.562,A -85,B 0,C 180,E1 -10139.723,E2 -10139.723} C_VEL
LIN {X 0,Y 417.93,Z 435.71,A -85,B 0,C 180,E1 -10143.033,E2 -10143.033} C_VEL
LIN {X 0,Y 417.624,Z 440.814,A -85,B 0,C 180,E1 -10146.179,E2 -10146.179} C_VEL
LIN {X 0,Y 417.524,Z 444.309,A -85,B 0,C 180,E1 -10148.265,E2 -10148.265} C_VEL
LIN {X 0,Y 417.316,Z 449.553,A -85,B 0,C 180,E1 -10151.338,E2 -10151.338} C_VEL
LIN {X 0,Y 417.253,Z 451.992,A -85,B 0,C 180,E1 -10152.73,E2 -10152.73} C_VEL
LIN {X 0,Y 420.02,Z 466.694,A -85,B 0,C 180,E1 -10153.323,E2 -10153.323} C_VEL
LIN {X 0,Y 421.747,Z 478.249,A -85,B 0,C 180,E1 -10153.95,E2 -10153.95} C_VEL
LIN {X 0,Y 421.207,Z 489.237,A -85,B 0,C 180,E1 -10154.64,E2 -10154.64} C_VEL
LIN {X 0,Y 420.65,Z 498.519,A -85,B 0,C 180,E1 -10155.363,E2 -10155.363} C_VEL
LIN {X 0,Y 420.066,Z 507.283,A -85,B 0,C 180,E1 -10156.187,E2 -10156.187} C_VEL
LIN {X 0,Y 419.485,Z 516.004,A -85,B 0,C 180,E1 -10157.174,E2 -10157.174} C_VEL
LIN {X 0,Y 418.907,Z 523.226,A -85,B 0,C 180,E1 -10158.14,E2 -10158.14} C_VEL
LIN {X 0,Y 418.426,Z 529.43,A -85,B 0,C 180,E1 -10159.108,E2 -10159.108} C_VEL
LIN {X 0,Y 417.976,Z 535.971,A -85,B 0,C 180,E1 -10160.32,E2 -10160.32} C_VEL
LIN {X 0,Y 417.695,Z 540.475,A -85,B 0,C 180,E1 -10161.29,E2 -10161.29} C_VEL
LIN {X 0,Y 417.366,Z 545.968,A -85,B 0,C 180,E1 -10162.745,E2 -10162.745} C_VEL
LIN {X 0,Y 417.163,Z 550.293,A -85,B 0,C 180,E1 -10164.198,E2 -10164.198} C_VEL
LIN {X 0,Y 417.15,Z 552.662,A -85,B 0,C 180,E1 -10165.168,E2 -10165.168} C_VEL
LIN {X 0,Y 417.024,Z 555.845,A -85,B 0,C 180,E1 -10167.102,E2 -10167.102} C_VEL
LIN {X 0,Y 417.053,Z 556.904,A -85,B 0,C 180,E1 -10168.068,E2 -10168.068} C_VEL
LIN {X 0,Y 416.993,Z 557.491,A -85,B 0,C 180,E1 -10169.034,E2 -10169.034} C_VEL
LIN {X 0,Y 416.993,Z 557.491,A -85,B 0,C 180,E1 -10170.965,E2 -10170.965} C_VEL
LIN {X 0,Y 417.053,Z 556.905,A -85,B 0,C 180,E1 -10171.931,E2 -10171.931} C_VEL
LIN {X 0,Y 417.023,Z 554.459,A -85,B 0,C 180,E1 -10173.865,E2 -10173.865} C_VEL
LIN {X 0,Y 417.164,Z 551.512,A -85,B 0,C 180,E1 -10175.316,E2 -10175.316} C_VEL
LIN {X 0,Y 417.277,Z 547.523,A -85,B 0,C 180,E1 -10176.77,E2 -10176.77} C_VEL
LIN {X 0,Y 417.55,Z 542.392,A -85,B 0,C 180,E1 -10178.225,E2 -10178.225} C_VEL
LIN {X 0,Y 417.893,Z 537.129,A -85,B 0,C 180,E1 -10179.437,E2 -10179.437} C_VEL
LIN {X 0,Y 418.317,Z 530.809,A -85,B 0,C 180,E1 -10180.65,E2 -10180.65} C_VEL
LIN {X 0,Y 418.761,Z 524.856,A -85,B 0,C 180,E1 -10181.618,E2 -10181.618} C_VEL
LIN {X 0,Y 419.337,Z 517.928,A -85,B 0,C 180,E1 -10182.584,E2 -10182.584} C_VEL
LIN {X 0,Y 419.883,Z 509.743,A -85,B 0,C 180,E1 -10183.552,E2 -10183.552} C_VEL
LIN {X 0,Y 420.443,Z 500.888,A -85,B 0,C 180,E1 -10184.428,E2 -10184.428} C_VEL
LIN {X 0,Y 420.995,Z 492.508,A -85,B 0,C 180,E1 -10185.119,E2 -10185.119} C_VEL
LIN {X 0,Y 421.517,Z 483.973,A -85,B 0,C 180,E1 -10185.706,E2 -10185.706} C_VEL
LIN {X 0,Y 421.638,Z 477.235,A -85,B 0,C 180,E1 -10186.112,E2 -10186.112} C_VEL
LIN {X 0,Y 419.615,Z 464.422,A -85,B 0,C 180,E1 -10186.775,E2 -10186.775} C_VEL
LIN {X 0,Y 417.464,Z 453.58,A -85,B 0,C 180,E1 -10187.207,E2 -10187.207} C_VEL
LIN {X 0,Y 417.252,Z 451.992,A -85,B 0,C 180,E1 -10187.269,E2 -10187.269} C_VEL
LIN {X 0,Y 417.45,Z 446.032,A -85,B 0,C 180,E1 -10190.704,E2 -10190.704} C_VEL
LIN {X 0,Y 417.576,Z 442.533,A -85,B 0,C 180,E1 -10192.774,E2 -10192.774} C_VEL
LIN {X 0,Y 417.788,Z 437.363,A -85,B 0,C 180,E1 -10195.936,E2 -10195.936} C_VEL
LIN {X 0,Y 418.09,Z 432.242,A -85,B 0,C 180,E1 -10199.175,E2 -10199.175} C_VEL
LIN {X 0,Y 418.414,Z 427.203,A -85,B 0,C 180,E1 -10202.513,E2 -10202.513} C_VEL
LIN {X 0,Y 418.797,Z 422.283,A -85,B 0,C 180,E1 -10205.968,E2 -10205.968} C_VEL
LIN {X 0,Y 419.106,Z 419.059,A -85,B 0,C 180,E1 -10208.348,E2 -10208.348} C_VEL
LIN {X 0,Y 419.376,Z 415.574,A -85,B 0,C 180,E1 -10211.051,E2 -10211.051} C_VEL
LIN {X 0,Y 419.205,Z 412.26,A -85,B 0,C 180,E1 -10213.871,E2 -10213.871} C_VEL
LIN {X 0,Y 418.79,Z 409.375,A -85,B 0,C 180,E1 -10216.524,E2 -10216.524} C_VEL
LIN {X 0,Y 418.384,Z 406.784,A -85,B 0,C 180,E1 -10219.104,E2 -10219.104} C_VEL
LIN {X 0,Y 418.255,Z 405.887,A -85,B 0,C 180,E1 -10220.618,E2 -10220.618} C_VEL
LIN {X 0,Y 418.243,Z 405.888,A -85,B 0,C 180,E1 -10223.975,E2 -10223.975} C_VEL
LIN {X 0,Y 418.258,Z 405.885,A -85,B 0,C 180,E1 -10227.154,E2 -10227.154} C_VEL
LIN {X 0,Y 418.272,Z 405.887,A -85,B 0,C 180,E1 -10230.838,E2 -10230.838} C_VEL
LIN {X 0,Y 418.267,Z 405.88,A -85,B 0,C 180,E1 -10234.095,E2 -10234.095} C_VEL
LIN {X 0,Y 418.233,Z 405.886,A -85,B 0,C 180,E1 -10237.263,E2 -10237.263} C_VEL
LIN {X 0,Y 418.278,Z 405.882,A -85,B 0,C 180,E1 -10240.363,E2 -10240.363} C_VEL
LIN {X 0,Y 418.312,Z 405.875,A -85,B 0,C 180,E1 -10243.404,E2 -10243.404} C_VEL
LIN {X 0,Y 418.341,Z 405.873,A -85,B 0,C 180,E1 -10246.999,E2 -10246.999} C_VEL
LIN {X 0,Y 418.335,Z 405.876,A -85,B 0,C 180,E1 -10250.328,E2 -10250.328} C_VEL
LIN {X 0,Y 418.507,Z 405.854,A -85,B 0,C 180,E1 -10252.279,E2 -10252.279} C_VEL
LIN {X 0,Y 418.507,Z 405.854,A -85,B 0,C 180,E1 -10254.217,E2 -10254.217} C_VEL
LIN {X 0,Y 418.539,Z 405.849,A -85,B 0,C 180,E1 -10258.075,E2 -10258.075} C_VEL
LIN {X 0,Y 418.666,Z 405.833,A -85,B 0,C 180,E1 -10259.999,E2 -10259.999} C_VEL
LIN {X 0,Y 418.505,Z 405.852,A -85,B 0,C 180,E1 -10262.887,E2 -10262.887} C_VEL
LIN {X 0,Y 418.487,Z 405.854,A -85,B 0,C 180,E1 -10266.751,E2 -10266.751} C_VEL
LIN {X 0,Y 418.393,Z 405.866,A -85,B 0,C 180,E1 -10268.695,E2 -10268.695} C_VEL
LIN {X 0,Y 418.308,Z 405.876,A -85,B 0,C 180,E1 -10271.631,E2 -10271.631} C_VEL
LIN {X 0,Y 418.299,Z 405.878,A -85,B 0,C 180,E1 -10274.597,E2 -10274.597} C_VEL
LIN {X 0,Y 418.281,Z 405.88,A -85,B 0,C 180,E1 -10277.603,E2 -10277.603} C_VEL
LIN {X 0,Y 418.242,Z 405.884,A -85,B 0,C 180,E1 -10280.663,E2 -10280.663} C_VEL
LIN {X 0,Y 418.281,Z 405.882,A -85,B 0,C 180,E1 -10283.781,E2 -10283.781} C_VEL
LIN {X 0,Y 418.303,Z 405.875,A -85,B 0,C 180,E1 -10287.07,E2 -10287.07} C_VEL
LIN {X 0,Y 418.255,Z 405.884,A -85,B 0,C 180,E1 -10290.271,E2 -10290.271} C_VEL
LIN {X 0,Y 418.242,Z 405.888,A -85,B 0,C 180,E1 -10293.677,E2 -10293.677} C_VEL
LIN {X 0,Y 418.24,Z 405.884,A -85,B 0,C 180,E1 -10297.223,E2 -10297.223} C_VEL
LIN {X 0,Y 418.259,Z 405.887,A -85,B 0,C 180,E1 -10299.68,E2 -10299.68} C_VEL
LIN {X 0,Y 418.278,Z 405.88,A -85,B 0,C 180,E1 -10302.33,E2 -10302.33} C_VEL
LIN {X 0,Y 418.267,Z 405.881,A -85,B 0,C 180,E1 -10305.114,E2 -10305.114} C_VEL
LIN {X 0,Y 418.286,Z 405.883,A -85,B 0,C 180,E1 -10307.774,E2 -10307.774} C_VEL
LIN {X 0,Y 418.258,Z 405.888,A -85,B 0,C 180,E1 -10311.56,E2 -10311.56} C_VEL
LIN {X 0,Y 418.254,Z 405.884,A -85,B 0,C 180,E1 -10315.159,E2 -10315.159} C_VEL
LIN {X 0,Y 418.239,Z 405.89,A -85,B 0,C 180,E1 -10317.472,E2 -10317.472} C_VEL
LIN {X 0,Y 418.263,Z 405.882,A -85,B 0,C 180,E1 -10320.896,E2 -10320.896} C_VEL
LIN {X 0,Y 418.266,Z 405.881,A -85,B 0,C 180,E1 -10324.096,E2 -10324.096} C_VEL
LIN {X 0,Y 418.233,Z 405.89,A -85,B 0,C 180,E1 -10327.264,E2 -10327.264} C_VEL
LIN {X 0,Y 418.279,Z 405.879,A -85,B 0,C 180,E1 -10330.365,E2 -10330.365} C_VEL
LIN {X 0,Y 418.313,Z 405.88,A -85,B 0,C 180,E1 -10333.405,E2 -10333.405} C_VEL
LIN {X 0,Y 418.342,Z 405.877,A -85,B 0,C 180,E1 -10336.999,E2 -10336.999} C_VEL
LIN {X 0,Y 418.338,Z 405.876,A -85,B 0,C 180,E1 -10340.329,E2 -10340.329} C_VEL
LIN {X 0,Y 418.491,Z 405.857,A -85,B 0,C 180,E1 -10343.249,E2 -10343.249} C_VEL
LIN {X 0,Y 418.338,Z 405.877,A -85,B 0,C 180,E1 -10345.182,E2 -10345.182} C_VEL
LIN {X 0,Y 418.541,Z 405.849,A -85,B 0,C 180,E1 -10348.076,E2 -10348.076} C_VEL
LIN {X 0,Y 418.669,Z 405.835,A -85,B 0,C 180,E1 -10350,E2 -10350} C_VEL
LIN {X 0,Y 418.507,Z 405.855,A -85,B 0,C 180,E1 -10352.888,E2 -10352.888} C_VEL
LIN {X 0,Y 418.491,Z 405.857,A -85,B 0,C 180,E1 -10356.751,E2 -10356.751} C_VEL
LIN {X 0,Y 418.338,Z 405.876,A -85,B 0,C 180,E1 -10359.672,E2 -10359.672} C_VEL
LIN {X 0,Y 418.318,Z 405.878,A -85,B 0,C 180,E1 -10363.337,E2 -10363.337} C_VEL
LIN {X 0,Y 417.625,Z 405.965,A -85,B 0,C 180,E1 -10364.141,E2 -10364.141} C_VEL
LIN {X 0,Y 414.747,Z 406.323,A -85,B 0,C 180,E1 -10365.446,E2 -10365.446} C_VEL
LIN {X 0,Y 412.334,Z 406.624,A -85,B 0,C 180,E1 -10366.5,E2 -10366.5} C_VEL
LIN {X 0,Y 411.313,Z 406.751,A -85,B 0,C 180,E1 -10367.315,E2 -10367.315} C_VEL
LIN {X 0,Y 411.236,Z 406.759,A -85,B 0,C 180,E1 -10367.591,E2 -10367.591} C_VEL
LIN {X 0,Y 411.193,Z 406.764,A -85,B 0,C 180,E1 -10371.034,E2 -10371.034} C_VEL
LIN {X 0,Y 411.223,Z 406.76,A -85,B 0,C 180,E1 -10374.215,E2 -10374.215} C_VEL
LIN {X 0,Y 411.255,Z 406.753,A -85,B 0,C 180,E1 -10377.478,E2 -10377.478} C_VEL
LIN {X 0,Y 411.185,Z 406.765,A -85,B 0,C 180,E1 -10380.848,E2 -10380.848} C_VEL
LIN {X 0,Y 411.202,Z 406.765,A -85,B 0,C 180,E1 -10384.334,E2 -10384.334} C_VEL
LIN {X 0,Y 411.199,Z 406.762,A -85,B 0,C 180,E1 -10387.973,E2 -10387.973} C_VEL
LIN {X 0,Y 411.205,Z 406.759,A -85,B 0,C 180,E1 -10391.236,E2 -10391.236} C_VEL
LIN {X 0,Y 411.219,Z 406.763,A -85,B 0,C 180,E1 -10394.484,E2 -10394.484} C_VEL
LIN {X 0,Y 411.173,Z 406.77,A -85,B 0,C 180,E1 -10398.195,E2 -10398.195} C_VEL
LIN {X 0,Y 411.219,Z 406.759,A -85,B 0,C 180,E1 -10400.777,E2 -10400.777} C_VEL
LIN {X 0,Y 411.195,Z 406.764,A -85,B 0,C 180,E1 -10404.472,E2 -10404.472} C_VEL
LIN {X 0,Y 411.168,Z 406.77,A -85,B 0,C 180,E1 -10408.004,E2 -10408.004} C_VEL
LIN {X 0,Y 411.219,Z 406.759,A -85,B 0,C 180,E1 -10411.411,E2 -10411.411} C_VEL
LIN {X 0,Y 411.232,Z 406.757,A -85,B 0,C 180,E1 -10414.707,E2 -10414.707} C_VEL
LIN {X 0,Y 411.201,Z 406.767,A -85,B 0,C 180,E1 -10417.914,E2 -10417.914} C_VEL
LIN {X 0,Y 411.22,Z 406.758,A -85,B 0,C 180,E1 -10421.052,E2 -10421.052} C_VEL
LIN {X 0,Y 411.258,Z 406.757,A -85,B 0,C 180,E1 -10424.132,E2 -10424.132} C_VEL
LIN {X 0,Y 411.299,Z 406.749,A -85,B 0,C 180,E1 -10427.166,E2 -10427.166} C_VEL
LIN {X 0,Y 411.289,Z 406.752,A -85,B 0,C 180,E1 -10430.162,E2 -10430.162} C_VEL
LIN {X 0,Y 411.478,Z 406.728,A -85,B 0,C 180,E1 -10432.147,E2 -10432.147} C_VEL
LIN {X 0,Y 411.471,Z 406.729,A -85,B 0,C 180,E1 -10434.119,E2 -10434.119} C_VEL
LIN {X 0,Y 411.51,Z 406.724,A -85,B 0,C 180,E1 -10438.043,E2 -10438.043} C_VEL
LIN {X 0,Y 411.638,Z 406.708,A -85,B 0,C 180,E1 -10440.001,E2 -10440.001} C_VEL
LIN {X 0,Y 411.463,Z 406.728,A -85,B 0,C 180,E1 -10442.938,E2 -10442.938} C_VEL
LIN {X 0,Y 411.457,Z 406.729,A -85,B 0,C 180,E1 -10446.868,E2 -10446.868} C_VEL
LIN {X 0,Y 411.351,Z 406.742,A -85,B 0,C 180,E1 -10448.846,E2 -10448.846} C_VEL
LIN {X 0,Y 411.281,Z 406.753,A -85,B 0,C 180,E1 -10451.833,E2 -10451.833} C_VEL
LIN {X 0,Y 411.258,Z 406.754,A -85,B 0,C 180,E1 -10454.853,E2 -10454.853} C_VEL
LIN {X 0,Y 411.25,Z 406.755,A -85,B 0,C 180,E1 -10457.916,E2 -10457.916} C_VEL
LIN {X 0,Y 411.194,Z 406.765,A -85,B 0,C 180,E1 -10461.035,E2 -10461.035} C_VEL
LIN {X 0,Y 411.225,Z 406.757,A -85,B 0,C 180,E1 -10464.216,E2 -10464.216} C_VEL
LIN {X 0,Y 411.257,Z 406.757,A -85,B 0,C 180,E1 -10467.478,E2 -10467.478} C_VEL
LIN {X 0,Y 411.188,Z 406.765,A -85,B 0,C 180,E1 -10470.848,E2 -10470.848} C_VEL
LIN {X 0,Y 411.205,Z 406.76,A -85,B 0,C 180,E1 -10474.334,E2 -10474.334} C_VEL
LIN {X 0,Y 411.2,Z 406.765,A -85,B 0,C 180,E1 -10477.974,E2 -10477.974} C_VEL
LIN {X 0,Y 411.235,Z 406.89,A -85,B 0,C 180,E1 -10479.732,E2 -10479.732} C_VEL
LIN {X 0,Y 411.723,Z 410.115,A -85,B 0,C 180,E1 -10483.063,E2 -10483.063} C_VEL
LIN {X 0,Y 412.137,Z 412.944,A -85,B 0,C 180,E1 -10485.743,E2 -10485.743} C_VEL
LIN {X 0,Y 412.372,Z 416.187,A -85,B 0,C 180,E1 -10488.581,E2 -10488.581} C_VEL
LIN {X 0,Y 412.166,Z 419.052,A -85,B 0,C 180,E1 -10490.884,E2 -10490.884} C_VEL
LIN {X 0,Y 411.876,Z 422.279,A -85,B 0,C 180,E1 -10493.329,E2 -10493.329} C_VEL
LIN {X 0,Y 411.436,Z 427.165,A -85,B 0,C 180,E1 -10496.865,E2 -10496.865} C_VEL
LIN {X 0,Y 411.071,Z 432.179,A -85,B 0,C 180,E1 -10500.277,E2 -10500.277} C_VEL
LIN {X 0,Y 410.772,Z 437.263,A -85,B 0,C 180,E1 -10503.587,E2 -10503.587} C_VEL
LIN {X 0,Y 410.5,Z 442.42,A -85,B 0,C 180,E1 -10506.811,E2 -10506.811} C_VEL
LIN {X 0,Y 410.3,Z 447.636,A -85,B 0,C 180,E1 -10509.966,E2 -10509.966} C_VEL
LIN {X 0,Y 410.175,Z 451.99,A -85,B 0,C 180,E1 -10512.445,E2 -10512.445} C_VEL
LIN {X 0,Y 412.197,Z 462.344,A -85,B 0,C 180,E1 -10512.846,E2 -10512.846} C_VEL
LIN {X 0,Y 413.865,Z 472.221,A -85,B 0,C 180,E1 -10513.339,E2 -10513.339} C_VEL
LIN {X 0,Y 414.808,Z 478.659,A -85,B 0,C 180,E1 -10513.713,E2 -10513.713} C_VEL
LIN {X 0,Y 414.373,Z 489.026,A -85,B 0,C 180,E1 -10514.38,E2 -10514.38} C_VEL
LIN {X 0,Y 413.753,Z 498.307,A -85,B 0,C 180,E1 -10515.113,E2 -10515.113} C_VEL
LIN {X 0,Y 413.154,Z 507.071,A -85,B 0,C 180,E1 -10515.951,E2 -10515.951} C_VEL
LIN {X 0,Y 412.535,Z 515.792,A -85,B 0,C 180,E1 -10516.954,E2 -10516.954} C_VEL
LIN {X 0,Y 411.933,Z 523.014,A -85,B 0,C 180,E1 -10517.936,E2 -10517.936} C_VEL
LIN {X 0,Y 411.426,Z 529.218,A -85,B 0,C 180,E1 -10518.92,E2 -10518.92} C_VEL
LIN {X 0,Y 410.936,Z 535.758,A -85,B 0,C 180,E1 -10520.153,E2 -10520.153} C_VEL
LIN {X 0,Y 410.635,Z 540.262,A -85,B 0,C 180,E1 -10521.139,E2 -10521.139} C_VEL
LIN {X 0,Y 410.293,Z 545.756,A -85,B 0,C 180,E1 -10522.619,E2 -10522.619} C_VEL
LIN {X 0,Y 410.083,Z 550.081,A -85,B 0,C 180,E1 -10524.098,E2 -10524.098} C_VEL
LIN {X 0,Y 410.06,Z 552.45,A -85,B 0,C 180,E1 -10525.084,E2 -10525.084} C_VEL
LIN {X 0,Y 409.923,Z 555.634,A -85,B 0,C 180,E1 -10527.052,E2 -10527.052} C_VEL
LIN {X 0,Y 409.964,Z 556.693,A -85,B 0,C 180,E1 -10528.035,E2 -10528.035} C_VEL
LIN {X 0,Y 409.919,Z 557.28,A -85,B 0,C 180,E1 -10529.017,E2 -10529.017} C_VEL
LIN {X 0,Y 409.919,Z 557.281,A -85,B 0,C 180,E1 -10530.982,E2 -10530.982} C_VEL
LIN {X 0,Y 409.964,Z 556.693,A -85,B 0,C 180,E1 -10531.965,E2 -10531.965} C_VEL
LIN {X 0,Y 409.943,Z 554.247,A -85,B 0,C 180,E1 -10533.932,E2 -10533.932} C_VEL
LIN {X 0,Y 410.063,Z 551.3,A -85,B 0,C 180,E1 -10535.409,E2 -10535.409} C_VEL
LIN {X 0,Y 410.2,Z 547.311,A -85,B 0,C 180,E1 -10536.888,E2 -10536.888} C_VEL
LIN {X 0,Y 410.499,Z 542.18,A -85,B 0,C 180,E1 -10538.367,E2 -10538.367} C_VEL
LIN {X 0,Y 410.863,Z 536.917,A -85,B 0,C 180,E1 -10539.6,E2 -10539.6} C_VEL
LIN {X 0,Y 411.296,Z 530.596,A -85,B 0,C 180,E1 -10540.833,E2 -10540.833} C_VEL
LIN {X 0,Y 411.769,Z 524.643,A -85,B 0,C 180,E1 -10541.818,E2 -10541.818} C_VEL
LIN {X 0,Y 412.372,Z 517.715,A -85,B 0,C 180,E1 -10542.8,E2 -10542.8} C_VEL
LIN {X 0,Y 412.945,Z 509.531,A -85,B 0,C 180,E1 -10543.784,E2 -10543.784} C_VEL
LIN {X 0,Y 413.551,Z 500.807,A -85,B 0,C 180,E1 -10544.662,E2 -10544.662} C_VEL
LIN {X 0,Y 414.126,Z 492.296,A -85,B 0,C 180,E1 -10545.376,E2 -10545.376} C_VEL
LIN {X 0,Y 414.748,Z 482.204,A -85,B 0,C 180,E1 -10546.067,E2 -10546.067} C_VEL
LIN {X 0,Y 414.581,Z 476.718,A -85,B 0,C 180,E1 -10546.41,E2 -10546.41} C_VEL
LIN {X 0,Y 412.447,Z 463.722,A -85,B 0,C 180,E1 -10547.093,E2 -10547.093} C_VEL
LIN {X 0,Y 410.285,Z 452.891,A -85,B 0,C 180,E1 -10547.529,E2 -10547.529} C_VEL
LIN {X 0,Y 410.159,Z 451.808,A -85,B 0,C 180,E1 -10547.577,E2 -10547.577} C_VEL
LIN {X 0,Y 410.297,Z 447.596,A -85,B 0,C 180,E1 -10550.034,E2 -10550.034} C_VEL
LIN {X 0,Y 410.499,Z 442.404,A -85,B 0,C 180,E1 -10553.189,E2 -10553.189} C_VEL
LIN {X 0,Y 410.762,Z 437.252,A -85,B 0,C 180,E1 -10556.413,E2 -10556.413} C_VEL
LIN {X 0,Y 411.063,Z 432.157,A -85,B 0,C 180,E1 -10559.723,E2 -10559.723} C_VEL
LIN {X 0,Y 411.443,Z 427.105,A -85,B 0,C 180,E1 -10563.176,E2 -10563.176} C_VEL
LIN {X 0,Y 411.866,Z 422.27,A -85,B 0,C 180,E1 -10566.678,E2 -10566.678} C_VEL
LIN {X 0,Y 412.257,Z 418.052,A -85,B 0,C 180,E1 -10569.901,E2 -10569.901} C_VEL
LIN {X 0,Y 412.362,Z 415.902,A -85,B 0,C 180,E1 -10571.657,E2 -10571.657} C_VEL
LIN {X 0,Y 412.119,Z 412.831,A -85,B 0,C 180,E1 -10574.361,E2 -10574.361} C_VEL
LIN {X 0,Y 411.672,Z 409.823,A -85,B 0,C 180,E1 -10577.229,E2 -10577.229} C_VEL
LIN {X 0,Y 411.233,Z 406.887,A -85,B 0,C 180,E1 -10580.268,E2 -10580.268} C_VEL
LIN {X 0,Y 411.193,Z 406.768,A -85,B 0,C 180,E1 -10583.446,E2 -10583.446} C_VEL
LIN {X 0,Y 411.205,Z 406.767,A -85,B 0,C 180,E1 -10586.872,E2 -10586.872} C_VEL
LIN {X 0,Y 411.238,Z 406.76,A -85,B 0,C 180,E1 -10590.641,E2 -10590.641} C_VEL
LIN {X 0,Y 411.234,Z 406.756,A -85,B 0,C 180,E1 -10593.618,E2 -10593.618} C_VEL
LIN {X 0,Y 411.199,Z 406.766,A -85,B 0,C 180,E1 -10596.852,E2 -10596.852} C_VEL
LIN {X 0,Y 411.21,Z 406.76,A -85,B 0,C 180,E1 -10600.05,E2 -10600.05} C_VEL
LIN {X 0,Y 411.258,Z 406.755,A -85,B 0,C 180,E1 -10603.13,E2 -10603.13} C_VEL
LIN {X 0,Y 411.3,Z 406.751,A -85,B 0,C 180,E1 -10606.895,E2 -10606.895} C_VEL
LIN {X 0,Y 411.287,Z 406.752,A -85,B 0,C 180,E1 -10610.161,E2 -10610.161} C_VEL
LIN {X 0,Y 411.455,Z 406.729,A -85,B 0,C 180,E1 -10613.132,E2 -10613.132} C_VEL
LIN {X 0,Y 411.306,Z 406.748,A -85,B 0,C 180,E1 -10615.098,E2 -10615.098} C_VEL
LIN {X 0,Y 411.508,Z 406.725,A -85,B 0,C 180,E1 -10618.042,E2 -10618.042} C_VEL
LIN {X 0,Y 411.635,Z 406.709,A -85,B 0,C 180,E1 -10619.999,E2 -10619.999} C_VEL
LIN {X 0,Y 411.46,Z 406.729,A -85,B 0,C 180,E1 -10622.937,E2 -10622.937} C_VEL
LIN {X 0,Y 411.454,Z 406.73,A -85,B 0,C 180,E1 -10626.867,E2 -10626.867} C_VEL
LIN {X 0,Y 411.286,Z 406.752,A -85,B 0,C 180,E1 -10629.838,E2 -10629.838} C_VEL
LIN {X 0,Y 411.298,Z 406.748,A -85,B 0,C 180,E1 -10633.104,E2 -10633.104} C_VEL
LIN {X 0,Y 411.257,Z 406.753,A -85,B 0,C 180,E1 -10636.869,E2 -10636.869} C_VEL
LIN {X 0,Y 411.223,Z 406.763,A -85,B 0,C 180,E1 -10639.987,E2 -10639.987} C_VEL
LIN {X 0,Y 411.196,Z 406.761,A -85,B 0,C 180,E1 -10643.147,E2 -10643.147} C_VEL
LIN {X 0,Y 411.231,Z 406.759,A -85,B 0,C 180,E1 -10646.381,E2 -10646.381} C_VEL
LIN {X 0,Y 411.204,Z 406.764,A -85,B 0,C 180,E1 -10649.712,E2 -10649.712} C_VEL
LIN {X 0,Y 411.199,Z 406.761,A -85,B 0,C 180,E1 -10653.156,E2 -10653.156} C_VEL
LIN {X 0,Y 411.189,Z 406.762,A -85,B 0,C 180,E1 -10656.553,E2 -10656.553} C_VEL
LIN {X 0,Y 411.222,Z 406.764,A -85,B 0,C 180,E1 -10659.731,E2 -10659.731} C_VEL
LIN {X 0,Y 411.224,Z 406.758,A -85,B 0,C 180,E1 -10663.126,E2 -10663.126} C_VEL
LIN {X 0,Y 411.224,Z 406.762,A -85,B 0,C 180,E1 -10665.872,E2 -10665.872} C_VEL
LIN {X 0,Y 411.203,Z 406.76,A -85,B 0,C 180,E1 -10668.764,E2 -10668.764} C_VEL
LIN {X 0,Y 411.197,Z 406.763,A -85,B 0,C 180,E1 -10672.028,E2 -10672.028} C_VEL
LIN {X 0,Y 411.2,Z 406.766,A -85,B 0,C 180,E1 -10675.667,E2 -10675.667} C_VEL
LIN {X 0,Y 411.184,Z 406.766,A -85,B 0,C 180,E1 -10679.153,E2 -10679.153} C_VEL
LIN {X 0,Y 411.253,Z 406.753,A -85,B 0,C 180,E1 -10682.523,E2 -10682.523} C_VEL
LIN {X 0,Y 411.222,Z 406.76,A -85,B 0,C 180,E1 -10685.785,E2 -10685.785} C_VEL
LIN {X 0,Y 411.192,Z 406.764,A -85,B 0,C 180,E1 -10688.966,E2 -10688.966} C_VEL
LIN {X 0,Y 411.248,Z 406.758,A -85,B 0,C 180,E1 -10692.085,E2 -10692.085} C_VEL
LIN {X 0,Y 411.256,Z 406.76,A -85,B 0,C 180,E1 -10695.148,E2 -10695.148} C_VEL
LIN {X 0,Y 411.28,Z 406.752,A -85,B 0,C 180,E1 -10698.168,E2 -10698.168} C_VEL
LIN {X 0,Y 411.478,Z 406.73,A -85,B 0,C 180,E1 -10702.147,E2 -10702.147} C_VEL
LIN {X 0,Y 411.473,Z 406.731,A -85,B 0,C 180,E1 -10704.118,E2 -10704.118} C_VEL
LIN {X 0,Y 411.511,Z 406.725,A -85,B 0,C 180,E1 -10708.043,E2 -10708.043} C_VEL
LIN {X 0,Y 411.639,Z 406.711,A -85,B 0,C 180,E1 -10710,E2 -10710} C_VEL
LIN {X 0,Y 411.463,Z 406.733,A -85,B 0,C 180,E1 -10712.937,E2 -10712.937} C_VEL
LIN {X 0,Y 411.458,Z 406.733,A -85,B 0,C 180,E1 -10716.867,E2 -10716.867} C_VEL
LIN {X 0,Y 411.29,Z 406.754,A -85,B 0,C 180,E1 -10719.839,E2 -10719.839} C_VEL
LIN {X 0,Y 411.279,Z 406.755,A -85,B 0,C 180,E1 -10723.325,E2 -10723.325} C_VEL
LIN {X 0,Y 411.253,Z 406.76,A -85,B 0,C 180,E1 -10726.889,E2 -10726.889} C_VEL
LIN {X 0,Y 411.236,Z 406.759,A -85,B 0,C 180,E1 -10727.591,E2 -10727.591} C_VEL
LIN {X 0,Y 410.576,Z 406.844,A -85,B 0,C 180,E1 -10728.409,E2 -10728.409} C_VEL
LIN {X 0,Y 407.688,Z 407.199,A -85,B 0,C 180,E1 -10729.737,E2 -10729.737} C_VEL
LIN {X 0,Y 405.244,Z 407.508,A -85,B 0,C 180,E1 -10730.81,E2 -10730.81} C_VEL
LIN {X 0,Y 404.208,Z 407.632,A -85,B 0,C 180,E1 -10731.64,E2 -10731.64} C_VEL
LIN {X 0,Y 404.132,Z 407.641,A -85,B 0,C 180,E1 -10731.921,E2 -10731.921} C_VEL
LIN {X 0,Y 404.212,Z 407.631,A -85,B 0,C 180,E1 -10735.297,E2 -10735.297} C_VEL
LIN {X 0,Y 404.192,Z 407.634,A -85,B 0,C 180,E1 -10738,E2 -10738} C_VEL
LIN {X 0,Y 404.135,Z 407.64,A -85,B 0,C 180,E1 -10741.558,E2 -10741.558} C_VEL
LIN {X 0,Y 404.181,Z 407.636,A -85,B 0,C 180,E1 -10745.016,E2 -10745.016} C_VEL
LIN {X 0,Y 404.158,Z 407.64,A -85,B 0,C 180,E1 -10748.756,E2 -10748.756} C_VEL
LIN {X 0,Y 404.187,Z 407.634,A -85,B 0,C 180,E1 -10751.611,E2 -10751.611} C_VEL
LIN {X 0,Y 404.184,Z 407.639,A -85,B 0,C 180,E1 -10754.529,E2 -10754.529} C_VEL
LIN {X 0,Y 404.132,Z 407.641,A -85,B 0,C 180,E1 -10757.296,E2 -10757.296} C_VEL
LIN {X 0,Y 404.164,Z 407.64,A -85,B 0,C 180,E1 -10759.956,E2 -10759.956} C_VEL
LIN {X 0,Y 404.135,Z 407.64,A -85,B 0,C 180,E1 -10763.125,E2 -10763.125} C_VEL
LIN {X 0,Y 404.14,Z 407.646,A -85,B 0,C 180,E1 -10766.188,E2 -10766.188} C_VEL
LIN {X 0,Y 404.151,Z 407.641,A -85,B 0,C 180,E1 -10769.716,E2 -10769.716} C_VEL
LIN {X 0,Y 404.191,Z 407.633,A -85,B 0,C 180,E1 -10773.123,E2 -10773.123} C_VEL
LIN {X 0,Y 404.173,Z 407.636,A -85,B 0,C 180,E1 -10775.335,E2 -10775.335} C_VEL
LIN {X 0,Y 404.134,Z 407.641,A -85,B 0,C 180,E1 -10778.581,E2 -10778.581} C_VEL
LIN {X 0,Y 404.206,Z 407.637,A -85,B 0,C 180,E1 -10781.762,E2 -10781.762} C_VEL
LIN {X 0,Y 404.207,Z 407.631,A -85,B 0,C 180,E1 -10784.883,E2 -10784.883} C_VEL
LIN {X 0,Y 404.252,Z 407.631,A -85,B 0,C 180,E1 -10787.959,E2 -10787.959} C_VEL
LIN {X 0,Y 404.43,Z 407.606,A -85,B 0,C 180,E1 -10792.1,E2 -10792.1} C_VEL
LIN {X 0,Y 404.42,Z 407.608,A -85,B 0,C 180,E1 -10794.016,E2 -10794.016} C_VEL
LIN {X 0,Y 404.479,Z 407.6,A -85,B 0,C 180,E1 -10798.009,E2 -10798.009} C_VEL
LIN {X 0,Y 404.608,Z 407.584,A -85,B 0,C 180,E1 -10800.001,E2 -10800.001} C_VEL
LIN {X 0,Y 404.42,Z 407.606,A -85,B 0,C 180,E1 -10802.989,E2 -10802.989} C_VEL
LIN {X 0,Y 404.409,Z 407.608,A -85,B 0,C 180,E1 -10806.988,E2 -10806.988} C_VEL
LIN {X 0,Y 404.255,Z 407.627,A -85,B 0,C 180,E1 -10810.012,E2 -10810.012} C_VEL
LIN {X 0,Y 404.264,Z 407.629,A -85,B 0,C 180,E1 -10813.212,E2 -10813.212} C_VEL
LIN {X 0,Y 404.214,Z 407.634,A -85,B 0,C 180,E1 -10817.008,E2 -10817.008} C_VEL
LIN {X 0,Y 404.162,Z 407.637,A -85,B 0,C 180,E1 -10820.352,E2 -10820.352} C_VEL
LIN {X 0,Y 404.168,Z 407.639,A -85,B 0,C 180,E1 -10823.575,E2 -10823.575} C_VEL
LIN {X 0,Y 404.182,Z 407.636,A -85,B 0,C 180,E1 -10825.767,E2 -10825.767} C_VEL
LIN {X 0,Y 404.194,Z 407.633,A -85,B 0,C 180,E1 -10828,E2 -10828} C_VEL
LIN {X 0,Y 404.138,Z 407.642,A -85,B 0,C 180,E1 -10831.559,E2 -10831.559} C_VEL
LIN {X 0,Y 404.185,Z 407.641,A -85,B 0,C 180,E1 -10835.017,E2 -10835.017} C_VEL
LIN {X 0,Y 404.158,Z 407.644,A -85,B 0,C 180,E1 -10838.757,E2 -10838.757} C_VEL
LIN {X 0,Y 404.287,Z 408.426,A -85,B 0,C 180,E1 -10840.104,E2 -10840.104} C_VEL
LIN {X 0,Y 404.752,Z 411.371,A -85,B 0,C 180,E1 -10843.175,E2 -10843.175} C_VEL
LIN {X 0,Y 405.222,Z 415.149,A -85,B 0,C 180,E1 -10846.756,E2 -10846.756} C_VEL
LIN {X 0,Y 405.319,Z 417.5,A -85,B 0,C 180,E1 -10848.785,E2 -10848.785} C_VEL
LIN {X 0,Y 405.08,Z 420.638,A -85,B 0,C 180,E1 -10851.349,E2 -10851.349} C_VEL
LIN {X 0,Y 404.606,Z 425.478,A -85,B 0,C 180,E1 -10855.026,E2 -10855.026} C_VEL
LIN {X 0,Y 404.197,Z 430.421,A -85,B 0,C 180,E1 -10858.559,E2 -10858.559} C_VEL
LIN {X 0,Y 403.849,Z 435.453,A -85,B 0,C 180,E1 -10861.974,E2 -10861.974} C_VEL
LIN {X 0,Y 403.575,Z 440.557,A -85,B 0,C 180,E1 -10865.295,E2 -10865.295} C_VEL
LIN {X 0,Y 403.317,Z 445.715,A -85,B 0,C 180,E1 -10868.535,E2 -10868.535} C_VEL
LIN {X 0,Y 403.085,Z 450.926,A -85,B 0,C 180,E1 -10871.709,E2 -10871.709} C_VEL
LIN {X 0,Y 403.097,Z 451.653,A -85,B 0,C 180,E1 -10872.122,E2 -10872.122} C_VEL
LIN {X 0,Y 405.186,Z 462.436,A -85,B 0,C 180,E1 -10872.552,E2 -10872.552} C_VEL
LIN {X 0,Y 406.983,Z 473.089,A -85,B 0,C 180,E1 -10873.103,E2 -10873.103} C_VEL
LIN {X 0,Y 407.973,Z 480.654,A -85,B 0,C 180,E1 -10873.574,E2 -10873.574} C_VEL
LIN {X 0,Y 407.395,Z 490.446,A -85,B 0,C 180,E1 -10874.234,E2 -10874.234} C_VEL
LIN {X 0,Y 406.761,Z 499.447,A -85,B 0,C 180,E1 -10874.979,E2 -10874.979} C_VEL
LIN {X 0,Y 406.209,Z 506.539,A -85,B 0,C 180,E1 -10875.67,E2 -10875.67} C_VEL
LIN {X 0,Y 405.572,Z 515.579,A -85,B 0,C 180,E1 -10876.726,E2 -10876.726} C_VEL
LIN {X 0,Y 404.94,Z 522.801,A -85,B 0,C 180,E1 -10877.725,E2 -10877.725} C_VEL
LIN {X 0,Y 404.435,Z 529.006,A -85,B 0,C 180,E1 -10878.726,E2 -10878.726} C_VEL
LIN {X 0,Y 403.915,Z 535.546,A -85,B 0,C 180,E1 -10879.98,E2 -10879.98} C_VEL
LIN {X 0,Y 403.598,Z 540.05,A -85,B 0,C 180,E1 -10880.983,E2 -10880.983} C_VEL
LIN {X 0,Y 403.214,Z 545.543,A -85,B 0,C 180,E1 -10882.488,E2 -10882.488} C_VEL
LIN {X 0,Y 402.992,Z 549.869,A -85,B 0,C 180,E1 -10883.994,E2 -10883.994} C_VEL
LIN {X 0,Y 402.972,Z 552.238,A -85,B 0,C 180,E1 -10884.997,E2 -10884.997} C_VEL
LIN {X 0,Y 402.865,Z 554.035,A -85,B 0,C 180,E1 -10885.998,E2 -10885.998} C_VEL
LIN {X 0,Y 402.862,Z 556.482,A -85,B 0,C 180,E1 -10888,E2 -10888} C_VEL
LIN {X 0,Y 402.847,Z 557.07,A -85,B 0,C 180,E1 -10889,E2 -10889} C_VEL
LIN {X 0,Y 402.847,Z 557.07,A -85,B 0,C 180,E1 -10890.999,E2 -10890.999} C_VEL
LIN {X 0,Y 402.862,Z 556.482,A -85,B 0,C 180,E1 -10891.999,E2 -10891.999} C_VEL
LIN {X 0,Y 402.865,Z 554.036,A -85,B 0,C 180,E1 -10894.001,E2 -10894.001} C_VEL
LIN {X 0,Y 402.966,Z 551.088,A -85,B 0,C 180,E1 -10895.504,E2 -10895.504} C_VEL
LIN {X 0,Y 403.119,Z 547.099,A -85,B 0,C 180,E1 -10897.009,E2 -10897.009} C_VEL
LIN {X 0,Y 403.435,Z 541.968,A -85,B 0,C 180,E1 -10898.515,E2 -10898.515} C_VEL
LIN {X 0,Y 403.838,Z 536.705,A -85,B 0,C 180,E1 -10899.769,E2 -10899.769} C_VEL
LIN {X 0,Y 404.285,Z 530.384,A -85,B 0,C 180,E1 -10901.024,E2 -10901.024} C_VEL
LIN {X 0,Y 404.794,Z 524.431,A -85,B 0,C 180,E1 -10902.025,E2 -10902.025} C_VEL
LIN {X 0,Y 405.417,Z 517.503,A -85,B 0,C 180,E1 -10903.024,E2 -10903.024} C_VEL
LIN {X 0,Y 406.024,Z 509.318,A -85,B 0,C 180,E1 -10904.024,E2 -10904.024} C_VEL
LIN {X 0,Y 406.653,Z 500.721,A -85,B 0,C 180,E1 -10904.904,E2 -10904.904} C_VEL
LIN {X 0,Y 407.26,Z 492.084,A -85,B 0,C 180,E1 -10905.642,E2 -10905.642} C_VEL
LIN {X 0,Y 407.905,Z 482.336,A -85,B 0,C 180,E1 -10906.322,E2 -10906.322} C_VEL
LIN {X 0,Y 407.666,Z 477.276,A -85,B 0,C 180,E1 -10906.653,E2 -10906.653} C_VEL
LIN {X 0,Y 405.492,Z 463.911,A -85,B 0,C 180,E1 -10907.38,E2 -10907.38} C_VEL
LIN {X 0,Y 403.248,Z 452.915,A -85,B 0,C 180,E1 -10907.839,E2 -10907.839} C_VEL
LIN {X 0,Y 403.089,Z 451.628,A -85,B 0,C 180,E1 -10907.893,E2 -10907.893} C_VEL
LIN {X 0,Y 403.248,Z 447.438,A -85,B 0,C 180,E1 -10910.399,E2 -10910.399} C_VEL
LIN {X 0,Y 403.446,Z 442.259,A -85,B 0,C 180,E1 -10913.619,E2 -10913.619} C_VEL
LIN {X 0,Y 403.74,Z 437.137,A -85,B 0,C 180,E1 -10916.909,E2 -10916.909} C_VEL
LIN {X 0,Y 404.047,Z 432.084,A -85,B 0,C 180,E1 -10920.293,E2 -10920.293} C_VEL
LIN {X 0,Y 404.443,Z 427.127,A -85,B 0,C 180,E1 -10923.783,E2 -10923.783} C_VEL
LIN {X 0,Y 404.9,Z 422.252,A -85,B 0,C 180,E1 -10927.409,E2 -10927.409} C_VEL
LIN {X 0,Y 405.236,Z 418.653,A -85,B 0,C 180,E1 -10930.262,E2 -10930.262} C_VEL
LIN {X 0,Y 405.297,Z 415.934,A -85,B 0,C 180,E1 -10932.552,E2 -10932.552} C_VEL
LIN {X 0,Y 404.925,Z 412.861,A -85,B 0,C 180,E1 -10935.365,E2 -10935.365} C_VEL
LIN {X 0,Y 404.445,Z 409.587,A -85,B 0,C 180,E1 -10938.675,E2 -10938.675} C_VEL
LIN {X 0,Y 404.265,Z 408.374,A -85,B 0,C 180,E1 -10939.966,E2 -10939.966} C_VEL
LIN {X 0,Y 404.155,Z 407.644,A -85,B 0,C 180,E1 -10941.491,E2 -10941.491} C_VEL
LIN {X 0,Y 404.183,Z 407.641,A -85,B 0,C 180,E1 -10944.983,E2 -10944.983} C_VEL
LIN {X 0,Y 404.148,Z 407.642,A -85,B 0,C 180,E1 -10948.554,E2 -10948.554} C_VEL
LIN {X 0,Y 404.194,Z 407.633,A -85,B 0,C 180,E1 -10952,E2 -10952} C_VEL
LIN {X 0,Y 404.173,Z 407.637,A -85,B 0,C 180,E1 -10955.334,E2 -10955.334} C_VEL
LIN {X 0,Y 404.134,Z 407.646,A -85,B 0,C 180,E1 -10958.58,E2 -10958.58} C_VEL
LIN {X 0,Y 404.205,Z 407.631,A -85,B 0,C 180,E1 -10961.761,E2 -10961.761} C_VEL
LIN {X 0,Y 404.201,Z 407.636,A -85,B 0,C 180,E1 -10964.881,E2 -10964.881} C_VEL
LIN {X 0,Y 404.251,Z 407.627,A -85,B 0,C 180,E1 -10967.958,E2 -10967.958} C_VEL
LIN {X 0,Y 404.428,Z 407.606,A -85,B 0,C 180,E1 -10972.099,E2 -10972.099} C_VEL
LIN {X 0,Y 404.418,Z 407.607,A -85,B 0,C 180,E1 -10974.014,E2 -10974.014} C_VEL
LIN {X 0,Y 404.477,Z 407.6,A -85,B 0,C 180,E1 -10978.008,E2 -10978.008} C_VEL
LIN {X 0,Y 404.605,Z 407.584,A -85,B 0,C 180,E1 -10979.999,E2 -10979.999} C_VEL
LIN {X 0,Y 404.417,Z 407.606,A -85,B 0,C 180,E1 -10982.988,E2 -10982.988} C_VEL
LIN {X 0,Y 404.405,Z 407.607,A -85,B 0,C 180,E1 -10986.987,E2 -10986.987} C_VEL
LIN {X 0,Y 404.252,Z 407.63,A -85,B 0,C 180,E1 -10990.011,E2 -10990.011} C_VEL
LIN {X 0,Y 404.259,Z 407.625,A -85,B 0,C 180,E1 -10993.211,E2 -10993.211} C_VEL
LIN {X 0,Y 404.211,Z 407.631,A -85,B 0,C 180,E1 -10997.008,E2 -10997.008} C_VEL
LIN {X 0,Y 404.156,Z 407.641,A -85,B 0,C 180,E1 -11000.351,E2 -11000.351} C_VEL
LIN {X 0,Y 404.162,Z 407.639,A -85,B 0,C 180,E1 -11003.574,E2 -11003.574} C_VEL
LIN {X 0,Y 404.176,Z 407.639,A -85,B 0,C 180,E1 -11005.766,E2 -11005.766} C_VEL
LIN {X 0,Y 404.191,Z 407.64,A -85,B 0,C 180,E1 -11007.999,E2 -11007.999} C_VEL
LIN {X 0,Y 404.14,Z 407.643,A -85,B 0,C 180,E1 -11011.56,E2 -11011.56} C_VEL
LIN {X 0,Y 404.178,Z 407.635,A -85,B 0,C 180,E1 -11015.016,E2 -11015.016} C_VEL
LIN {X 0,Y 404.157,Z 407.637,A -85,B 0,C 180,E1 -11018.756,E2 -11018.756} C_VEL
LIN {X 0,Y 404.185,Z 407.64,A -85,B 0,C 180,E1 -11021.611,E2 -11021.611} C_VEL
LIN {X 0,Y 404.194,Z 407.633,A -85,B 0,C 180,E1 -11024.53,E2 -11024.53} C_VEL
LIN {X 0,Y 404.2,Z 407.635,A -85,B 0,C 180,E1 -11027.305,E2 -11027.305} C_VEL
LIN {X 0,Y 404.162,Z 407.64,A -85,B 0,C 180,E1 -11029.956,E2 -11029.956} C_VEL
LIN {X 0,Y 404.134,Z 407.643,A -85,B 0,C 180,E1 -11033.124,E2 -11033.124} C_VEL
LIN {X 0,Y 404.139,Z 407.64,A -85,B 0,C 180,E1 -11036.188,E2 -11036.188} C_VEL
LIN {X 0,Y 404.14,Z 407.644,A -85,B 0,C 180,E1 -11039.715,E2 -11039.715} C_VEL
LIN {X 0,Y 404.19,Z 407.637,A -85,B 0,C 180,E1 -11043.123,E2 -11043.123} C_VEL
LIN {X 0,Y 404.173,Z 407.642,A -85,B 0,C 180,E1 -11045.335,E2 -11045.335} C_VEL
LIN {X 0,Y 404.134,Z 407.641,A -85,B 0,C 180,E1 -11048.581,E2 -11048.581} C_VEL
LIN {X 0,Y 404.206,Z 407.636,A -85,B 0,C 180,E1 -11051.762,E2 -11051.762} C_VEL
LIN {X 0,Y 404.202,Z 407.638,A -85,B 0,C 180,E1 -11054.882,E2 -11054.882} C_VEL
LIN {X 0,Y 404.253,Z 407.627,A -85,B 0,C 180,E1 -11057.959,E2 -11057.959} C_VEL
LIN {X 0,Y 404.429,Z 407.608,A -85,B 0,C 180,E1 -11062.1,E2 -11062.1} C_VEL
LIN {X 0,Y 404.421,Z 407.61,A -85,B 0,C 180,E1 -11064.015,E2 -11064.015} C_VEL
LIN {X 0,Y 404.479,Z 407.601,A -85,B 0,C 180,E1 -11068.009,E2 -11068.009} C_VEL
LIN {X 0,Y 404.608,Z 407.587,A -85,B 0,C 180,E1 -11070,E2 -11070} C_VEL
LIN {X 0,Y 404.42,Z 407.61,A -85,B 0,C 180,E1 -11072.989,E2 -11072.989} C_VEL
LIN {X 0,Y 404.409,Z 407.611,A -85,B 0,C 180,E1 -11076.987,E2 -11076.987} C_VEL
LIN {X 0,Y 404.255,Z 407.631,A -85,B 0,C 180,E1 -11080.012,E2 -11080.012} C_VEL
LIN {X 0,Y 404.263,Z 407.631,A -85,B 0,C 180,E1 -11083.212,E2 -11083.212} C_VEL
LIN {X 0,Y 404.212,Z 407.637,A -85,B 0,C 180,E1 -11087.007,E2 -11087.007} C_VEL
LIN {X 0,Y 404.16,Z 407.64,A -85,B 0,C 180,E1 -11090.352,E2 -11090.352} C_VEL
LIN {X 0,Y 404.132,Z 407.641,A -85,B 0,C 180,E1 -11091.921,E2 -11091.921} C_VEL
LIN {X 0,Y 403.49,Z 407.726,A -85,B 0,C 180,E1 -11092.753,E2 -11092.753} C_VEL
LIN {X 0,Y 400.658,Z 408.084,A -85,B 0,C 180,E1 -11094.105,E2 -11094.105} C_VEL
LIN {X 0,Y 398.248,Z 408.383,A -85,B 0,C 180,E1 -11095.197,E2 -11095.197} C_VEL
LIN {X 0,Y 397.214,Z 408.507,A -85,B 0,C 180,E1 -11096.041,E2 -11096.041} C_VEL
LIN {X 0,Y 397.13,Z 408.515,A -85,B 0,C 180,E1 -11096.327,E2 -11096.327} C_VEL
LIN {X 0,Y 397.119,Z 408.521,A -85,B 0,C 180,E1 -11098.544,E2 -11098.544} C_VEL
LIN {X 0,Y 397.074,Z 408.522,A -85,B 0,C 180,E1 -11102.072,E2 -11102.072} C_VEL
LIN {X 0,Y 397.116,Z 408.515,A -85,B 0,C 180,E1 -11105.504,E2 -11105.504} C_VEL
LIN {X 0,Y 397.132,Z 408.515,A -85,B 0,C 180,E1 -11108.863,E2 -11108.863} C_VEL
LIN {X 0,Y 397.154,Z 408.516,A -85,B 0,C 180,E1 -11112.256,E2 -11112.256} C_VEL
LIN {X 0,Y 397.106,Z 408.516,A -85,B 0,C 180,E1 -11115.066,E2 -11115.066} C_VEL
LIN {X 0,Y 397.062,Z 408.526,A -85,B 0,C 180,E1 -11118.021,E2 -11118.021} C_VEL
LIN {X 0,Y 397.129,Z 408.513,A -85,B 0,C 180,E1 -11121.138,E2 -11121.138} C_VEL
LIN {X 0,Y 397.115,Z 408.518,A -85,B 0,C 180,E1 -11124.497,E2 -11124.497} C_VEL
LIN {X 0,Y 397.107,Z 408.521,A -85,B 0,C 180,E1 -11127.932,E2 -11127.932} C_VEL
LIN {X 0,Y 397.122,Z 408.515,A -85,B 0,C 180,E1 -11131.457,E2 -11131.457} C_VEL
LIN {X 0,Y 397.148,Z 408.512,A -85,B 0,C 180,E1 -11134.488,E2 -11134.488} C_VEL
LIN {X 0,Y 397.104,Z 408.516,A -85,B 0,C 180,E1 -11137.086,E2 -11137.086} C_VEL
LIN {X 0,Y 397.144,Z 408.513,A -85,B 0,C 180,E1 -11140.353,E2 -11140.353} C_VEL
LIN {X 0,Y 397.166,Z 408.512,A -85,B 0,C 180,E1 -11143.554,E2 -11143.554} C_VEL
LIN {X 0,Y 397.224,Z 408.501,A -85,B 0,C 180,E1 -11146.703,E2 -11146.703} C_VEL
LIN {X 0,Y 397.214,Z 408.509,A -85,B 0,C 180,E1 -11149.809,E2 -11149.809} C_VEL
LIN {X 0,Y 397.36,Z 408.484,A -85,B 0,C 180,E1 -11152.889,E2 -11152.889} C_VEL
LIN {X 0,Y 397.252,Z 408.498,A -85,B 0,C 180,E1 -11154.926,E2 -11154.926} C_VEL
LIN {X 0,Y 397.448,Z 408.476,A -85,B 0,C 180,E1 -11157.974,E2 -11157.974} C_VEL
LIN {X 0,Y 397.577,Z 408.46,A -85,B 0,C 180,E1 -11160.001,E2 -11160.001} C_VEL
LIN {X 0,Y 397.378,Z 408.483,A -85,B 0,C 180,E1 -11163.042,E2 -11163.042} C_VEL
LIN {X 0,Y 397.361,Z 408.487,A -85,B 0,C 180,E1 -11167.112,E2 -11167.112} C_VEL
LIN {X 0,Y 397.215,Z 408.503,A -85,B 0,C 180,E1 -11170.192,E2 -11170.192} C_VEL
LIN {X 0,Y 397.224,Z 408.507,A -85,B 0,C 180,E1 -11173.322,E2 -11173.322} C_VEL
LIN {X 0,Y 397.18,Z 408.511,A -85,B 0,C 180,E1 -11177.156,E2 -11177.156} C_VEL
LIN {X 0,Y 397.101,Z 408.518,A -85,B 0,C 180,E1 -11180.731,E2 -11180.731} C_VEL
LIN {X 0,Y 397.131,Z 408.513,A -85,B 0,C 180,E1 -11184.019,E2 -11184.019} C_VEL
LIN {X 0,Y 397.193,Z 408.51,A -85,B 0,C 180,E1 -11187.391,E2 -11187.391} C_VEL
LIN {X 0,Y 397.078,Z 408.523,A -85,B 0,C 180,E1 -11190.883,E2 -11190.883} C_VEL
LIN {X 0,Y 397.125,Z 408.515,A -85,B 0,C 180,E1 -11194.494,E2 -11194.494} C_VEL
LIN {X 0,Y 397.106,Z 408.522,A -85,B 0,C 180,E1 -11198.275,E2 -11198.275} C_VEL
LIN {X 0,Y 397.118,Z 408.521,A -85,B 0,C 180,E1 -11198.86,E2 -11198.86} C_VEL
LIN {X 0,Y 397.583,Z 411.578,A -85,B 0,C 180,E1 -11202.201,E2 -11202.201} C_VEL
LIN {X 0,Y 397.978,Z 414.434,A -85,B 0,C 180,E1 -11205.06,E2 -11205.06} C_VEL
LIN {X 0,Y 398.317,Z 417.508,A -85,B 0,C 180,E1 -11207.896,E2 -11207.896} C_VEL
LIN {X 0,Y 398.064,Z 421.163,A -85,B 0,C 180,E1 -11210.973,E2 -11210.973} C_VEL
LIN {X 0,Y 397.632,Z 425.538,A -85,B 0,C 180,E1 -11214.394,E2 -11214.394} C_VEL
LIN {X 0,Y 397.184,Z 430.35,A -85,B 0,C 180,E1 -11217.938,E2 -11217.938} C_VEL
LIN {X 0,Y 396.83,Z 435.351,A -85,B 0,C 180,E1 -11221.434,E2 -11221.434} C_VEL
LIN {X 0,Y 396.532,Z 440.425,A -85,B 0,C 180,E1 -11224.826,E2 -11224.826} C_VEL
LIN {X 0,Y 396.275,Z 445.555,A -85,B 0,C 180,E1 -11228.134,E2 -11228.134} C_VEL
LIN {X 0,Y 396.02,Z 450.739,A -85,B 0,C 180,E1 -11231.371,E2 -11231.371} C_VEL
LIN {X 0,Y 396.023,Z 451.582,A -85,B 0,C 180,E1 -11231.796,E2 -11231.796} C_VEL
LIN {X 0,Y 398.068,Z 462.027,A -85,B 0,C 180,E1 -11232.222,E2 -11232.222} C_VEL
LIN {X 0,Y 399.863,Z 472.099,A -85,B 0,C 180,E1 -11232.754,E2 -11232.754} C_VEL
LIN {X 0,Y 401.045,Z 480.829,A -85,B 0,C 180,E1 -11233.307,E2 -11233.307} C_VEL
LIN {X 0,Y 400.699,Z 488.603,A -85,B 0,C 180,E1 -11233.833,E2 -11233.833} C_VEL
LIN {X 0,Y 399.991,Z 497.883,A -85,B 0,C 180,E1 -11234.588,E2 -11234.588} C_VEL
LIN {X 0,Y 399.251,Z 507.116,A -85,B 0,C 180,E1 -11235.505,E2 -11235.505} C_VEL
LIN {X 0,Y 398.626,Z 515.367,A -85,B 0,C 180,E1 -11236.491,E2 -11236.491} C_VEL
LIN {X 0,Y 397.98,Z 522.589,A -85,B 0,C 180,E1 -11237.507,E2 -11237.507} C_VEL
LIN {X 0,Y 397.439,Z 528.793,A -85,B 0,C 180,E1 -11238.525,E2 -11238.525} C_VEL
LIN {X 0,Y 396.911,Z 535.334,A -85,B 0,C 180,E1 -11239.801,E2 -11239.801} C_VEL
LIN {X 0,Y 396.56,Z 539.838,A -85,B 0,C 180,E1 -11240.822,E2 -11240.822} C_VEL
LIN {X 0,Y 396.164,Z 545.332,A -85,B 0,C 180,E1 -11242.354,E2 -11242.354} C_VEL
LIN {X 0,Y 395.912,Z 549.657,A -85,B 0,C 180,E1 -11243.886,E2 -11243.886} C_VEL
LIN {X 0,Y 395.884,Z 552.027,A -85,B 0,C 180,E1 -11244.907,E2 -11244.907} C_VEL
LIN {X 0,Y 395.789,Z 553.824,A -85,B 0,C 180,E1 -11245.927,E2 -11245.927} C_VEL
LIN {X 0,Y 395.76,Z 556.27,A -85,B 0,C 180,E1 -11247.964,E2 -11247.964} C_VEL
LIN {X 0,Y 395.777,Z 556.859,A -85,B 0,C 180,E1 -11248.982,E2 -11248.982} C_VEL
LIN {X 0,Y 395.777,Z 556.86,A -85,B 0,C 180,E1 -11251.017,E2 -11251.017} C_VEL
LIN {X 0,Y 395.76,Z 556.271,A -85,B 0,C 180,E1 -11252.035,E2 -11252.035} C_VEL
LIN {X 0,Y 395.789,Z 553.825,A -85,B 0,C 180,E1 -11254.073,E2 -11254.073} C_VEL
LIN {X 0,Y 395.87,Z 550.876,A -85,B 0,C 180,E1 -11255.603,E2 -11255.603} C_VEL
LIN {X 0,Y 396.064,Z 546.887,A -85,B 0,C 180,E1 -11257.135,E2 -11257.135} C_VEL
LIN {X 0,Y 396.391,Z 541.756,A -85,B 0,C 180,E1 -11258.667,E2 -11258.667} C_VEL
LIN {X 0,Y 396.803,Z 536.492,A -85,B 0,C 180,E1 -11259.944,E2 -11259.944} C_VEL
LIN {X 0,Y 397.284,Z 530.171,A -85,B 0,C 180,E1 -11261.22,E2 -11261.22} C_VEL
LIN {X 0,Y 397.817,Z 524.219,A -85,B 0,C 180,E1 -11262.239,E2 -11262.239} C_VEL
LIN {X 0,Y 398.465,Z 517.29,A -85,B 0,C 180,E1 -11263.255,E2 -11263.255} C_VEL
LIN {X 0,Y 399.117,Z 509.106,A -85,B 0,C 180,E1 -11264.271,E2 -11264.271} C_VEL
LIN {X 0,Y 399.746,Z 500.726,A -85,B 0,C 180,E1 -11265.147,E2 -11265.147} C_VEL
LIN {X 0,Y 400.397,Z 491.872,A -85,B 0,C 180,E1 -11265.917,E2 -11265.917} C_VEL
LIN {X 0,Y 401.047,Z 482.416,A -85,B 0,C 180,E1 -11266.59,E2 -11266.59} C_VEL
LIN {X 0,Y 400.304,Z 474.829,A -85,B 0,C 180,E1 -11267.088,E2 -11267.088} C_VEL
LIN {X 0,Y 398.307,Z 463.188,A -85,B 0,C 180,E1 -11267.723,E2 -11267.723} C_VEL
LIN {X 0,Y 396.076,Z 452.272,A -85,B 0,C 180,E1 -11268.184,E2 -11268.184} C_VEL
LIN {X 0,Y 396.023,Z 451.442,A -85,B 0,C 180,E1 -11268.223,E2 -11268.223} C_VEL
LIN {X 0,Y 396.171,Z 447.268,A -85,B 0,C 180,E1 -11270.78,E2 -11270.78} C_VEL
LIN {X 0,Y 396.36,Z 443.829,A -85,B 0,C 180,E1 -11272.959,E2 -11272.959} C_VEL
LIN {X 0,Y 396.612,Z 438.719,A -85,B 0,C 180,E1 -11276.295,E2 -11276.295} C_VEL
LIN {X 0,Y 396.964,Z 433.517,A -85,B 0,C 180,E1 -11279.828,E2 -11279.828} C_VEL
LIN {X 0,Y 397.319,Z 428.711,A -85,B 0,C 180,E1 -11283.253,E2 -11283.253} C_VEL
LIN {X 0,Y 397.796,Z 423.823,A -85,B 0,C 180,E1 -11286.918,E2 -11286.918} C_VEL
LIN {X 0,Y 398.109,Z 420.632,A -85,B 0,C 180,E1 -11289.458,E2 -11289.458} C_VEL
LIN {X 0,Y 398.293,Z 417.432,A -85,B 0,C 180,E1 -11292.174,E2 -11292.174} C_VEL
LIN {X 0,Y 397.955,Z 414.297,A -85,B 0,C 180,E1 -11295.056,E2 -11295.056} C_VEL
LIN {X 0,Y 397.533,Z 411.423,A -85,B 0,C 180,E1 -11297.945,E2 -11297.945} C_VEL
LIN {X 0,Y 397.115,Z 408.521,A -85,B 0,C 180,E1 -11301.14,E2 -11301.14} C_VEL
LIN {X 0,Y 397.117,Z 408.52,A -85,B 0,C 180,E1 -11304.496,E2 -11304.496} C_VEL
LIN {X 0,Y 397.109,Z 408.515,A -85,B 0,C 180,E1 -11307.931,E2 -11307.931} C_VEL
LIN {X 0,Y 397.123,Z 408.515,A -85,B 0,C 180,E1 -11311.456,E2 -11311.456} C_VEL
LIN {X 0,Y 397.149,Z 408.514,A -85,B 0,C 180,E1 -11314.487,E2 -11314.487} C_VEL
LIN {X 0,Y 397.105,Z 408.519,A -85,B 0,C 180,E1 -11317.085,E2 -11317.085} C_VEL
LIN {X 0,Y 397.143,Z 408.514,A -85,B 0,C 180,E1 -11320.352,E2 -11320.352} C_VEL
LIN {X 0,Y 397.161,Z 408.509,A -85,B 0,C 180,E1 -11323.552,E2 -11323.552} C_VEL
LIN {X 0,Y 397.223,Z 408.507,A -85,B 0,C 180,E1 -11326.702,E2 -11326.702} C_VEL
LIN {X 0,Y 397.212,Z 408.503,A -85,B 0,C 180,E1 -11329.808,E2 -11329.808} C_VEL
LIN {X 0,Y 397.358,Z 408.487,A -85,B 0,C 180,E1 -11332.888,E2 -11332.888} C_VEL
LIN {X 0,Y 397.25,Z 408.5,A -85,B 0,C 180,E1 -11334.925,E2 -11334.925} C_VEL
LIN {X 0,Y 397.446,Z 408.476,A -85,B 0,C 180,E1 -11337.973,E2 -11337.973} C_VEL
LIN {X 0,Y 397.574,Z 408.46,A -85,B 0,C 180,E1 -11339.999,E2 -11339.999} C_VEL
LIN {X 0,Y 397.376,Z 408.483,A -85,B 0,C 180,E1 -11343.041,E2 -11343.041} C_VEL
LIN {X 0,Y 397.357,Z 408.485,A -85,B 0,C 180,E1 -11347.111,E2 -11347.111} C_VEL
LIN {X 0,Y 397.211,Z 408.509,A -85,B 0,C 180,E1 -11350.191,E2 -11350.191} C_VEL
LIN {X 0,Y 397.219,Z 408.502,A -85,B 0,C 180,E1 -11353.321,E2 -11353.321} C_VEL
LIN {X 0,Y 397.164,Z 408.512,A -85,B 0,C 180,E1 -11356.446,E2 -11356.446} C_VEL
LIN {X 0,Y 397.141,Z 408.514,A -85,B 0,C 180,E1 -11359.647,E2 -11359.647} C_VEL
LIN {X 0,Y 397.128,Z 408.513,A -85,B 0,C 180,E1 -11363.04,E2 -11363.04} C_VEL
LIN {X 0,Y 397.128,Z 408.517,A -85,B 0,C 180,E1 -11366.258,E2 -11366.258} C_VEL
LIN {X 0,Y 397.119,Z 408.515,A -85,B 0,C 180,E1 -11368.543,E2 -11368.543} C_VEL
LIN {X 0,Y 397.104,Z 408.521,A -85,B 0,C 180,E1 -11372.068,E2 -11372.068} C_VEL
LIN {X 0,Y 397.113,Z 408.518,A -85,B 0,C 180,E1 -11375.504,E2 -11375.504} C_VEL
LIN {X 0,Y 397.131,Z 408.513,A -85,B 0,C 180,E1 -11378.863,E2 -11378.863} C_VEL
LIN {X 0,Y 397.153,Z 408.512,A -85,B 0,C 180,E1 -11382.255,E2 -11382.255} C_VEL
LIN {X 0,Y 397.143,Z 408.512,A -85,B 0,C 180,E1 -11385.06,E2 -11385.06} C_VEL
LIN {X 0,Y 397.149,Z 408.513,A -85,B 0,C 180,E1 -11388.007,E2 -11388.007} C_VEL
LIN {X 0,Y 397.103,Z 408.522,A -85,B 0,C 180,E1 -11391.726,E2 -11391.726} C_VEL
LIN {X 0,Y 397.12,Z 408.521,A -85,B 0,C 180,E1 -11395.507,E2 -11395.507} C_VEL
LIN {X 0,Y 397.073,Z 408.523,A -85,B 0,C 180,E1 -11399.118,E2 -11399.118} C_VEL
LIN {X 0,Y 397.189,Z 408.506,A -85,B 0,C 180,E1 -11402.61,E2 -11402.61} C_VEL
LIN {X 0,Y 397.128,Z 408.514,A -85,B 0,C 180,E1 -11405.982,E2 -11405.982} C_VEL
LIN {X 0,Y 397.134,Z 408.518,A -85,B 0,C 180,E1 -11409.705,E2 -11409.705} C_VEL
LIN {X 0,Y 397.177,Z 408.513,A -85,B 0,C 180,E1 -11412.845,E2 -11412.845} C_VEL
LIN {X 0,Y 397.224,Z 408.507,A -85,B 0,C 180,E1 -11416.703,E2 -11416.703} C_VEL
LIN {X 0,Y 397.214,Z 408.508,A -85,B 0,C 180,E1 -11419.809,E2 -11419.809} C_VEL
LIN {X 0,Y 397.361,Z 408.489,A -85,B 0,C 180,E1 -11422.888,E2 -11422.888} C_VEL
LIN {X 0,Y 397.253,Z 408.504,A -85,B 0,C 180,E1 -11424.925,E2 -11424.925} C_VEL
LIN {X 0,Y 397.448,Z 408.477,A -85,B 0,C 180,E1 -11427.974,E2 -11427.974} C_VEL
LIN {X 0,Y 397.577,Z 408.463,A -85,B 0,C 180,E1 -11430,E2 -11430} C_VEL
LIN {X 0,Y 397.378,Z 408.487,A -85,B 0,C 180,E1 -11433.042,E2 -11433.042} C_VEL
LIN {X 0,Y 397.361,Z 408.489,A -85,B 0,C 180,E1 -11437.112,E2 -11437.112} C_VEL
LIN {X 0,Y 397.215,Z 408.508,A -85,B 0,C 180,E1 -11440.191,E2 -11440.191} C_VEL
LIN {X 0,Y 397.223,Z 408.507,A -85,B 0,C 180,E1 -11443.321,E2 -11443.321} C_VEL
LIN {X 0,Y 397.178,Z 408.513,A -85,B 0,C 180,E1 -11447.155,E2 -11447.155} C_VEL
LIN {X 0,Y 397.099,Z 408.523,A -85,B 0,C 180,E1 -11450.73,E2 -11450.73} C_VEL
LIN {X 0,Y 397.129,Z 408.514,A -85,B 0,C 180,E1 -11454.018,E2 -11454.018} C_VEL
LIN {X 0,Y 397.13,Z 408.515,A -85,B 0,C 180,E1 -11456.327,E2 -11456.327} C_VEL
LIN {X 0,Y 396.461,Z 408.598,A -85,B 0,C 180,E1 -11457.174,E2 -11457.174} C_VEL
LIN {X 0,Y 393.586,Z 408.961,A -85,B 0,C 180,E1 -11458.549,E2 -11458.549} C_VEL
LIN {X 0,Y 391.147,Z 409.264,A -85,B 0,C 180,E1 -11459.66,E2 -11459.66} C_VEL
LIN {X 0,Y 390.095,Z 409.396,A -85,B 0,C 180,E1 -11460.52,E2 -11460.52} C_VEL
LIN {X 0,Y 390.007,Z 409.4,A -85,B 0,C 180,E1 -11460.812,E2 -11460.812} C_VEL
LIN {X 0,Y 390.064,Z 409.395,A -85,B 0,C 180,E1 -11464.025,E2 -11464.025} C_VEL
LIN {X 0,Y 390.042,Z 409.396,A -85,B 0,C 180,E1 -11467.552,E2 -11467.552} C_VEL
LIN {X 0,Y 390.078,Z 409.393,A -85,B 0,C 180,E1 -11470.826,E2 -11470.826} C_VEL
LIN {X 0,Y 390.097,Z 409.391,A -85,B 0,C 180,E1 -11473.894,E2 -11473.894} C_VEL
LIN {X 0,Y 390.038,Z 409.397,A -85,B 0,C 180,E1 -11477.626,E2 -11477.626} C_VEL
LIN {X 0,Y 390.088,Z 409.391,A -85,B 0,C 180,E1 -11480.908,E2 -11480.908} C_VEL
LIN {X 0,Y 390.081,Z 409.392,A -85,B 0,C 180,E1 -11484.793,E2 -11484.793} C_VEL
LIN {X 0,Y 390.043,Z 409.398,A -85,B 0,C 180,E1 -11488.498,E2 -11488.498} C_VEL
LIN {X 0,Y 390.113,Z 409.394,A -85,B 0,C 180,E1 -11492.07,E2 -11492.07} C_VEL
LIN {X 0,Y 390.075,Z 409.394,A -85,B 0,C 180,E1 -11495.52,E2 -11495.52} C_VEL
LIN {X 0,Y 390.051,Z 409.395,A -85,B 0,C 180,E1 -11498.878,E2 -11498.878} C_VEL
LIN {X 0,Y 390.124,Z 409.389,A -85,B 0,C 180,E1 -11502.167,E2 -11502.167} C_VEL
LIN {X 0,Y 390.142,Z 409.385,A -85,B 0,C 180,E1 -11505.393,E2 -11505.393} C_VEL
LIN {X 0,Y 390.144,Z 409.383,A -85,B 0,C 180,E1 -11508.572,E2 -11508.572} C_VEL
LIN {X 0,Y 390.34,Z 409.363,A -85,B 0,C 180,E1 -11511.994,E2 -11511.994} C_VEL
LIN {X 0,Y 390.224,Z 409.373,A -85,B 0,C 180,E1 -11514.834,E2 -11514.834} C_VEL
LIN {X 0,Y 390.417,Z 409.353,A -85,B 0,C 180,E1 -11517.937,E2 -11517.937} C_VEL
LIN {X 0,Y 390.547,Z 409.336,A -85,B 0,C 180,E1 -11520.001,E2 -11520.001} C_VEL
LIN {X 0,Y 390.312,Z 409.364,A -85,B 0,C 180,E1 -11523.097,E2 -11523.097} C_VEL
LIN {X 0,Y 390.327,Z 409.361,A -85,B 0,C 180,E1 -11526.202,E2 -11526.202} C_VEL
LIN {X 0,Y 390.312,Z 409.362,A -85,B 0,C 180,E1 -11528.283,E2 -11528.283} C_VEL
LIN {X 0,Y 390.168,Z 409.38,A -85,B 0,C 180,E1 -11532.484,E2 -11532.484} C_VEL
LIN {X 0,Y 390.137,Z 409.387,A -85,B 0,C 180,E1 -11535.677,E2 -11535.677} C_VEL
LIN {X 0,Y 390.103,Z 409.391,A -85,B 0,C 180,E1 -11538.923,E2 -11538.923} C_VEL
LIN {X 0,Y 390.038,Z 409.396,A -85,B 0,C 180,E1 -11542.235,E2 -11542.235} C_VEL
LIN {X 0,Y 390.118,Z 409.388,A -85,B 0,C 180,E1 -11545.744,E2 -11545.744} C_VEL
LIN {X 0,Y 390.058,Z 409.4,A -85,B 0,C 180,E1 -11549.11,E2 -11549.11} C_VEL
LIN {X 0,Y 390.042,Z 409.398,A -85,B 0,C 180,E1 -11552.722,E2 -11552.722} C_VEL
LIN {X 0,Y 390.057,Z 409.398,A -85,B 0,C 180,E1 -11555.826,E2 -11555.826} C_VEL
LIN {X 0,Y 390.045,Z 409.401,A -85,B 0,C 180,E1 -11557.78,E2 -11557.78} C_VEL
LIN {X 0,Y 390.167,Z 410.032,A -85,B 0,C 180,E1 -11559.236,E2 -11559.236} C_VEL
LIN {X 0,Y 390.596,Z 412.967,A -85,B 0,C 180,E1 -11562.464,E2 -11562.464} C_VEL
LIN {X 0,Y 390.998,Z 415.975,A -85,B 0,C 180,E1 -11565.493,E2 -11565.493} C_VEL
LIN {X 0,Y 391.251,Z 419.054,A -85,B 0,C 180,E1 -11568.347,E2 -11568.347} C_VEL
LIN {X 0,Y 391.018,Z 422.216,A -85,B 0,C 180,E1 -11571.018,E2 -11571.018} C_VEL
LIN {X 0,Y 390.629,Z 425.999,A -85,B 0,C 180,E1 -11574.059,E2 -11574.059} C_VEL
LIN {X 0,Y 390.184,Z 430.278,A -85,B 0,C 180,E1 -11577.292,E2 -11577.292} C_VEL
LIN {X 0,Y 389.818,Z 435.248,A -85,B 0,C 180,E1 -11580.871,E2 -11580.871} C_VEL
LIN {X 0,Y 389.505,Z 440.454,A -85,B 0,C 180,E1 -11584.446,E2 -11584.446} C_VEL
LIN {X 0,Y 389.236,Z 445.396,A -85,B 0,C 180,E1 -11587.718,E2 -11587.718} C_VEL
LIN {X 0,Y 388.983,Z 450.554,A -85,B 0,C 180,E1 -11591.021,E2 -11591.021} C_VEL
LIN {X 0,Y 388.938,Z 451.305,A -85,B 0,C 180,E1 -11591.452,E2 -11591.452} C_VEL
LIN {X 0,Y 391.001,Z 461.403,A -85,B 0,C 180,E1 -11591.874,E2 -11591.874} C_VEL
LIN {X 0,Y 392.542,Z 470.513,A -85,B 0,C 180,E1 -11592.351,E2 -11592.351} C_VEL
LIN {X 0,Y 393.929,Z 479.492,A -85,B 0,C 180,E1 -11592.922,E2 -11592.922} C_VEL
LIN {X 0,Y 394.188,Z 483.962,A -85,B 0,C 180,E1 -11593.229,E2 -11593.229} C_VEL
LIN {X 0,Y 393.253,Z 496.319,A -85,B 0,C 180,E1 -11594.185,E2 -11594.185} C_VEL
LIN {X 0,Y 392.381,Z 506.624,A -85,B 0,C 180,E1 -11595.213,E2 -11595.213} C_VEL
LIN {X 0,Y 391.667,Z 515.18,A -85,B 0,C 180,E1 -11596.249,E2 -11596.249} C_VEL
LIN {X 0,Y 391.036,Z 522.377,A -85,B 0,C 180,E1 -11597.281,E2 -11597.281} C_VEL
LIN {X 0,Y 390.423,Z 528.58,A -85,B 0,C 180,E1 -11598.316,E2 -11598.316} C_VEL
LIN {X 0,Y 389.895,Z 535.122,A -85,B 0,C 180,E1 -11599.615,E2 -11599.615} C_VEL
LIN {X 0,Y 389.496,Z 539.625,A -85,B 0,C 180,E1 -11600.654,E2 -11600.654} C_VEL
LIN {X 0,Y 389.095,Z 545.119,A -85,B 0,C 180,E1 -11602.214,E2 -11602.214} C_VEL
LIN {X 0,Y 388.836,Z 549.445,A -85,B 0,C 180,E1 -11603.774,E2 -11603.774} C_VEL
LIN {X 0,Y 388.78,Z 551.814,A -85,B 0,C 180,E1 -11604.814,E2 -11604.814} C_VEL
LIN {X 0,Y 388.715,Z 553.613,A -85,B 0,C 180,E1 -11605.853,E2 -11605.853} C_VEL
LIN {X 0,Y 388.659,Z 556.059,A -85,B 0,C 180,E1 -11607.927,E2 -11607.927} C_VEL
LIN {X 0,Y 388.69,Z 556.648,A -85,B 0,C 180,E1 -11608.964,E2 -11608.964} C_VEL
LIN {X 0,Y 388.69,Z 556.649,A -85,B 0,C 180,E1 -11611.036,E2 -11611.036} C_VEL
LIN {X 0,Y 388.659,Z 556.059,A -85,B 0,C 180,E1 -11612.072,E2 -11612.072} C_VEL
LIN {X 0,Y 388.715,Z 553.614,A -85,B 0,C 180,E1 -11614.147,E2 -11614.147} C_VEL
LIN {X 0,Y 388.781,Z 551.815,A -85,B 0,C 180,E1 -11615.185,E2 -11615.185} C_VEL
LIN {X 0,Y 388.917,Z 548.207,A -85,B 0,C 180,E1 -11616.745,E2 -11616.745} C_VEL
LIN {X 0,Y 389.214,Z 543.46,A -85,B 0,C 180,E1 -11618.305,E2 -11618.305} C_VEL
LIN {X 0,Y 389.697,Z 537.436,A -85,B 0,C 180,E1 -11619.865,E2 -11619.865} C_VEL
LIN {X 0,Y 390.166,Z 531.336,A -85,B 0,C 180,E1 -11621.165,E2 -11621.165} C_VEL
LIN {X 0,Y 390.717,Z 525.634,A -85,B 0,C 180,E1 -11622.201,E2 -11622.201} C_VEL
LIN {X 0,Y 391.515,Z 517.078,A -85,B 0,C 180,E1 -11623.495,E2 -11623.495} C_VEL
LIN {X 0,Y 392.186,Z 508.893,A -85,B 0,C 180,E1 -11624.529,E2 -11624.529} C_VEL
LIN {X 0,Y 392.886,Z 500.514,A -85,B 0,C 180,E1 -11625.418,E2 -11625.418} C_VEL
LIN {X 0,Y 393.579,Z 491.66,A -85,B 0,C 180,E1 -11626.201,E2 -11626.201} C_VEL
LIN {X 0,Y 394.186,Z 482.479,A -85,B 0,C 180,E1 -11626.869,E2 -11626.869} C_VEL
LIN {X 0,Y 393.051,Z 473.247,A -85,B 0,C 180,E1 -11627.484,E2 -11627.484} C_VEL
LIN {X 0,Y 391.26,Z 462.86,A -85,B 0,C 180,E1 -11628.057,E2 -11628.057} C_VEL
LIN {X 0,Y 389.002,Z 452.05,A -85,B 0,C 180,E1 -11628.526,E2 -11628.526} C_VEL
LIN {X 0,Y 388.931,Z 451.255,A -85,B 0,C 180,E1 -11628.567,E2 -11628.567} C_VEL
LIN {X 0,Y 389.127,Z 447.079,A -85,B 0,C 180,E1 -11631.174,E2 -11631.174} C_VEL
LIN {X 0,Y 389.283,Z 443.667,A -85,B 0,C 180,E1 -11633.401,E2 -11633.401} C_VEL
LIN {X 0,Y 389.584,Z 438.602,A -85,B 0,C 180,E1 -11636.807,E2 -11636.807} C_VEL
LIN {X 0,Y 389.933,Z 433.589,A -85,B 0,C 180,E1 -11640.308,E2 -11640.308} C_VEL
LIN {X 0,Y 390.383,Z 428.425,A -85,B 0,C 180,E1 -11644.092,E2 -11644.092} C_VEL
LIN {X 0,Y 390.875,Z 423.78,A -85,B 0,C 180,E1 -11647.708,E2 -11647.708} C_VEL
LIN {X 0,Y 391.175,Z 420.625,A -85,B 0,C 180,E1 -11650.299,E2 -11650.299} C_VEL
LIN {X 0,Y 391.184,Z 417.498,A -85,B 0,C 180,E1 -11653.054,E2 -11653.054} C_VEL
LIN {X 0,Y 390.824,Z 414.448,A -85,B 0,C 180,E1 -11655.996,E2 -11655.996} C_VEL
LIN {X 0,Y 390.33,Z 411.056,A -85,B 0,C 180,E1 -11659.594,E2 -11659.594} C_VEL
LIN {X 0,Y 390.134,Z 409.907,A -85,B 0,C 180,E1 -11660.912,E2 -11660.912} C_VEL
LIN {X 0,Y 390.043,Z 409.401,A -85,B 0,C 180,E1 -11662.448,E2 -11662.448} C_VEL
LIN {X 0,Y 390.065,Z 409.396,A -85,B 0,C 180,E1 -11666.044,E2 -11666.044} C_VEL
LIN {X 0,Y 390.046,Z 409.398,A -85,B 0,C 180,E1 -11668.497,E2 -11668.497} C_VEL
LIN {X 0,Y 390.114,Z 409.387,A -85,B 0,C 180,E1 -11672.069,E2 -11672.069} C_VEL
LIN {X 0,Y 390.076,Z 409.392,A -85,B 0,C 180,E1 -11675.518,E2 -11675.518} C_VEL
LIN {X 0,Y 390.051,Z 409.4,A -85,B 0,C 180,E1 -11678.877,E2 -11678.877} C_VEL
LIN {X 0,Y 390.123,Z 409.387,A -85,B 0,C 180,E1 -11682.166,E2 -11682.166} C_VEL
LIN {X 0,Y 390.139,Z 409.384,A -85,B 0,C 180,E1 -11685.392,E2 -11685.392} C_VEL
LIN {X 0,Y 390.143,Z 409.39,A -85,B 0,C 180,E1 -11688.57,E2 -11688.57} C_VEL
LIN {X 0,Y 390.338,Z 409.361,A -85,B 0,C 180,E1 -11691.993,E2 -11691.993} C_VEL
LIN {X 0,Y 390.222,Z 409.376,A -85,B 0,C 180,E1 -11694.833,E2 -11694.833} C_VEL
LIN {X 0,Y 390.415,Z 409.351,A -85,B 0,C 180,E1 -11697.936,E2 -11697.936} C_VEL
LIN {X 0,Y 390.544,Z 409.336,A -85,B 0,C 180,E1 -11699.999,E2 -11699.999} C_VEL
LIN {X 0,Y 390.31,Z 409.363,A -85,B 0,C 180,E1 -11703.096,E2 -11703.096} C_VEL
LIN {X 0,Y 390.303,Z 409.365,A -85,B 0,C 180,E1 -11706.641,E2 -11706.641} C_VEL
LIN {X 0,Y 390.198,Z 409.376,A -85,B 0,C 180,E1 -11709.328,E2 -11709.328} C_VEL
LIN {X 0,Y 390.187,Z 409.378,A -85,B 0,C 180,E1 -11713.438,E2 -11713.438} C_VEL
LIN {X 0,Y 390.143,Z 409.383,A -85,B 0,C 180,E1 -11717.308,E2 -11717.308} C_VEL
LIN {X 0,Y 390.08,Z 409.394,A -85,B 0,C 180,E1 -11720.47,E2 -11720.47} C_VEL
LIN {X 0,Y 390.082,Z 409.392,A -85,B 0,C 180,E1 -11723.351,E2 -11723.351} C_VEL
LIN {X 0,Y 390.106,Z 409.388,A -85,B 0,C 180,E1 -11726.768,E2 -11726.768} C_VEL
LIN {X 0,Y 390.038,Z 409.399,A -85,B 0,C 180,E1 -11730.299,E2 -11730.299} C_VEL
LIN {X 0,Y 390.077,Z 409.397,A -85,B 0,C 180,E1 -11733.953,E2 -11733.953} C_VEL
LIN {X 0,Y 390.04,Z 409.4,A -85,B 0,C 180,E1 -11737.552,E2 -11737.552} C_VEL
LIN {X 0,Y 390.076,Z 409.392,A -85,B 0,C 180,E1 -11740.826,E2 -11740.826} C_VEL
LIN {X 0,Y 390.122,Z 409.391,A -85,B 0,C 180,E1 -11743.898,E2 -11743.898} C_VEL
LIN {X 0,Y 390.114,Z 409.393,A -85,B 0,C 180,E1 -11747.613,E2 -11747.613} C_VEL
LIN {X 0,Y 390.088,Z 409.391,A -85,B 0,C 180,E1 -11750.908,E2 -11750.908} C_VEL
LIN {X 0,Y 390.08,Z 409.392,A -85,B 0,C 180,E1 -11754.793,E2 -11754.793} C_VEL
LIN {X 0,Y 390.017,Z 409.399,A -85,B 0,C 180,E1 -11758.496,E2 -11758.496} C_VEL
LIN {X 0,Y 390.112,Z 409.388,A -85,B 0,C 180,E1 -11762.07,E2 -11762.07} C_VEL
LIN {X 0,Y 390.076,Z 409.397,A -85,B 0,C 180,E1 -11765.52,E2 -11765.52} C_VEL
LIN {X 0,Y 390.051,Z 409.397,A -85,B 0,C 180,E1 -11768.878,E2 -11768.878} C_VEL
LIN {X 0,Y 390.123,Z 409.39,A -85,B 0,C 180,E1 -11772.167,E2 -11772.167} C_VEL
LIN {X 0,Y 390.139,Z 409.391,A -85,B 0,C 180,E1 -11775.393,E2 -11775.393} C_VEL
LIN {X 0,Y 390.144,Z 409.387,A -85,B 0,C 180,E1 -11778.571,E2 -11778.571} C_VEL
LIN {X 0,Y 390.318,Z 409.368,A -85,B 0,C 180,E1 -11782.535,E2 -11782.535} C_VEL
LIN {X 0,Y 390.35,Z 409.577,A -85,B 0,C 180,E1 -11782.704,E2 -11782.704} C_VEL
LIN {X 0,Y 390.911,Z 411.475,A -85,B 0,C 180,E1 -11783.16,E2 -11783.16} C_VEL
LIN {X 0,Y 392.539,Z 413.757,A -85,B 0,C 180,E1 -11784.349,E2 -11784.349} C_VEL
LIN {X 0,Y 394.308,Z 415.018,A -85,B 0,C 180,E1 -11785.912,E2 -11785.912} C_VEL
LIN {X 0,Y 395.197,Z 415.231,A -85,B 0,C 180,E1 -11786.942,E2 -11786.942} C_VEL
LIN {X 0,Y 396.207,Z 415.463,A -85,B 0,C 180,E1 -11788.984,E2 -11788.984} C_VEL
LIN {X 0,Y 396.373,Z 415.461,A -85,B 0,C 180,E1 -11790,E2 -11790} C_VEL
LIN {X 0,Y 395.807,Z 415.384,A -85,B 0,C 180,E1 -11792.035,E2 -11792.035} C_VEL
LIN {X 0,Y 394.474,Z 415.059,A -85,B 0,C 180,E1 -11793.894,E2 -11793.894} C_VEL
LIN {X 0,Y 392.69,Z 413.905,A -85,B 0,C 180,E1 -11795.52,E2 -11795.52} C_VEL
LIN {X 0,Y 390.994,Z 411.648,A -85,B 0,C 180,E1 -11796.774,E2 -11796.774} C_VEL
LIN {X 0,Y 390.385,Z 409.728,A -85,B 0,C 180,E1 -11797.268,E2 -11797.268} C_VEL
LIN {X 0,Y 390.316,Z 409.368,A -85,B 0,C 180,E1 -11797.353,E2 -11797.353} C_VEL
LIN {X 0,Y 390.165,Z 409.385,A -85,B 0,C 180,E1 -11800.377,E2 -11800.377} C_VEL
LIN {X 0,Y 390.166,Z 409.385,A -85,B 0,C 180,E1 -11803.543,E2 -11803.543} C_VEL
LIN {X 0,Y 390.145,Z 409.388,A -85,B 0,C 180,E1 -11807.308,E2 -11807.308} C_VEL
LIN {X 0,Y 390.083,Z 409.395,A -85,B 0,C 180,E1 -11810.47,E2 -11810.47} C_VEL
LIN {X 0,Y 390.086,Z 409.391,A -85,B 0,C 180,E1 -11813.351,E2 -11813.351} C_VEL
LIN {X 0,Y 390.109,Z 409.392,A -85,B 0,C 180,E1 -11816.768,E2 -11816.768} C_VEL
LIN {X 0,Y 390.035,Z 409.401,A -85,B 0,C 180,E1 -11820.3,E2 -11820.3} C_VEL
LIN {X 0,Y 390.007,Z 409.4,A -85,B 0,C 180,E1 -11820.812,E2 -11820.812} C_VEL
LIN {X 0,Y 389.334,Z 409.485,A -85,B 0,C 180,E1 -11821.674,E2 -11821.674} C_VEL
LIN {X 0,Y 386.486,Z 409.84,A -85,B 0,C 180,E1 -11823.075,E2 -11823.075} C_VEL
LIN {X 0,Y 384.089,Z 410.141,A -85,B 0,C 180,E1 -11824.208,E2 -11824.208} C_VEL
LIN {X 0,Y 383.071,Z 410.266,A -85,B 0,C 180,E1 -11825.084,E2 -11825.084} C_VEL
LIN {X 0,Y 382.995,Z 410.274,A -85,B 0,C 180,E1 -11825.381,E2 -11825.381} C_VEL
LIN {X 0,Y 383.004,Z 410.277,A -85,B 0,C 180,E1 -11828.6,E2 -11828.6} C_VEL
LIN {X 0,Y 383.042,Z 410.268,A -85,B 0,C 180,E1 -11831.339,E2 -11831.339} C_VEL
LIN {X 0,Y 383.029,Z 410.276,A -85,B 0,C 180,E1 -11834.309,E2 -11834.309} C_VEL
LIN {X 0,Y 383.005,Z 410.272,A -85,B 0,C 180,E1 -11837.24,E2 -11837.24} C_VEL
